METHOD PUBLIC Cycle // cyclic call for checking XtsStation state masks and command input from process
//-------------------------------------------------------------------------------------------------
//-------------------------------------------------------------------------------------------------
//  HAUD 2024 10 21
//  cyclic call required
//
//-------------------------------------------------------------------------------------------------
//-------------------------------------------------------------------------------------------------
// reference checks
//-------------------------------------------------------------------------------------------------
IF NOT __ISVALIDREF(_stControl)
THEN
  _eCheck                           := E_PROCESS_CHECK.REFERENCE_CTRL_INVALID;
  RETURN;
END_IF

IF NOT __ISVALIDREF(_stState)
THEN
  _eCheck                           := E_PROCESS_CHECK.REFERENCE_STATE_INVALID;
  RETURN;
END_IF
//-------------------------------------------------------------------------------------------------
//-------------------------------------------------------------------------------------------------
// plausibility checks
//-------------------------------------------------------------------------------------------------
IF NOT Check()
THEN
  // you shall not pass!!
  RETURN;
END_IF
//-------------------------------------------------------------------------------------------------
//-------------------------------------------------------------------------------------------------
// Message device identification
//-------------------------------------------------------------------------------------------------
_stMsg.eDevice                      := e_Device.Process + TO_UINT(_nProcessId);
//-------------------------------------------------------------------------------------------------
//-------------------------------------------------------------------------------------------------
// XtsStation states:
//  - fb_ProcessCollector extends fb_StationCollector: 
//    --> cyclic call of States() for getting station masks
//
//  - sets bit for every XtsStation
//-------------------------------------------------------------------------------------------------
//
States();                           // not just mental, literal
//-------------------------------------------------------------------------------------------------
//-------------------------------------------------------------------------------------------------
// process states
//-------------------------------------------------------------------------------------------------
CASE _stState.State
OF
  //-----------------------------------------------------------------------------------------------
  E_PROCESS_STATE.PROCESS_DISABLE:  // default wait state
    //-------------------------------------------------------------------------
    CASE _eStateProgress            // check if all my XtsStations are disabled
    OF
      E_PROGRESS.PROGRESS_INIT:
        IF (_wStateDisable = EXPT(2,_nStationCount)-1)                  // all stations in process range must be disabled at this point
        THEN
          // on a sunny afternoon, nothing to do, just sit and wait
          _eStateProgress           := E_PROGRESS.PROGRESS_BUSY;

          IF (_MessageLevel > E_MessageType.eMessageInfo)
          THEN
            _stMsg.eType            := E_MessageType.eMessageVerbose;
            _stMsg.eSubdevice       := e_Subdevice.Process_ProcessCollector_Cycle;
            _stMsg.iErrorNumber     := _wStateDisable;
            _stMsg.sText            := concat('_wStateDisable: ', BitsToString(_wStateDisable));
            _stMsg.sText            := concat(_stMsg.sText, ': ');
            _stMsg.sText            := concat(_stMsg.sText, TO_STRING(_eStateProgress));
            f_MessageSet(_stMsg);
          END_IF
        END_IF
    END_CASE
    //-------------------------------------------------------------------------
    CASE _eStateProgress            // check for process enable signal
    OF
      E_PROGRESS.PROGRESS_BUSY:
      CASE _stControl.Cmd                                               // check process command
      OF
        E_PROCESS_CTRL.PROCESS_ENABLE:                                  // only one thing to say here..
          _eCmd                     := _stControl.Cmd;                  // copy command from interface to local switch
          // you do what I say, when I say it
          _wActivateStation         := _stControl.ActivateStation;      // on enabling of process, copy my active stations from interface

          LogControl(_eCmd);

          _eStateProgress           := E_PROGRESS.PROGRESS_INIT;        // switch back sub state
          _stState.State            := E_PROCESS_STATE.PROCESS_ENABLE;  // switch to enable

          IF (_MessageLevel > E_MessageType.eMessageError)
          THEN
            _stMsg.eType            := E_MessageType.eMessageInfo;
            _stMsg.eSubdevice       := e_Subdevice.Process_ProcessCollector_Cycle;
            _stMsg.iErrorNumber     := _nProcessId;
            _stMsg.sText            := concat(TO_STRING(_stState.State), ': ');
            _stMsg.sText            := concat(_stMsg.sText, TO_STRING(_eStateProgress));
            f_MessageSet(_stMsg);
          END_IF
      END_CASE
    END_CASE
END_CASE
//-------------------------------------------------------------------------------------------------
//-------------------------------------------------------------------------------------------------
CASE _stState.State
OF
  //-----------------------------------------------------------------------------------------------
  E_PROCESS_STATE.PROCESS_ENABLE:   // wait here for process command "allow infeed"
    //-------------------------------------------------------------------------
    CASE _eStateProgress
    OF
      E_PROGRESS.PROGRESS_INIT:
        IF (_wStateEnable = _wActivateStation)                          // all active stations must be enabled
        THEN
          // we are truly equal, yet not the same
          _eStateProgress           := E_PROGRESS.PROGRESS_BUSY;

          IF (_MessageLevel > E_MessageType.eMessageInfo)
          THEN
            _stMsg.eType            := E_MessageType.eMessageVerbose;
            _stMsg.eSubdevice       := e_Subdevice.Process_ProcessCollector_Cycle;
            _stMsg.iErrorNumber     := _wStateEnable;
            _stMsg.sText            := concat('_wStateEnable: ', BitsToString(_wStateEnable));
            _stMsg.sText            := concat(_stMsg.sText, ': ');
            _stMsg.sText            := concat(_stMsg.sText, TO_STRING(_eStateProgress));
            f_MessageSet(_stMsg);
          END_IF
        END_IF
    END_CASE
    //-------------------------------------------------------------------------
    CASE _eStateProgress
    OF
      E_PROGRESS.PROGRESS_BUSY:
      // check command for further instructions
      CASE _stControl.Cmd
      OF
        E_PROCESS_CTRL.PROCESS_DISABLE:                                 // command decided to switch OFF  
          _eCmd                     := _stControl.Cmd;                  // copy command from interface

          LogControl(_eCmd);

          _eStateProgress           := E_PROGRESS.PROGRESS_INIT;        // switch back sub state
          _stState.State            := E_PROCESS_STATE.PROCESS_DISABLE;

          IF (_MessageLevel > E_MessageType.eMessageInfo)
          THEN
            _stMsg.eType            := E_MessageType.eMessageVerbose;
            _stMsg.eSubdevice       := e_Subdevice.Process_ProcessCollector_Cycle;
            _stMsg.iErrorNumber     := _nProcessId;
            _stMsg.sText            := concat(TO_STRING(_stState.State), ': ');
            _stMsg.sText            := concat(_stMsg.sText, TO_STRING(_eStateProgress));
            f_MessageSet(_stMsg);
          END_IF


        E_PROCESS_CTRL.PROCESS_STATIONS_INFEED,
        E_PROCESS_CTRL.PROCESS_STATIONS_ENTER,
        E_PROCESS_CTRL.PROCESS_STATIONS_SEND:                           // command decided to allow checking the infeed into process
          _eStateProgress           := E_PROGRESS.PROGRESS_INIT;        // switch back sub state
          _stState.State            := E_PROCESS_STATE.PROCESS_STATIONS_INFEED;

          IF (_MessageLevel > E_MessageType.eMessageWarning)
          THEN
            _stMsg.eType            := E_MessageType.eMessageInfo;
            _stMsg.eSubdevice       := e_Subdevice.Process_ProcessCollector_Cycle;
            _stMsg.iErrorNumber     := _nProcessId;
            _stMsg.sText            := concat(TO_STRING(_stState.State), ': ');
            _stMsg.sText            := concat(_stMsg.sText, TO_STRING(_eStateProgress));
            f_MessageSet(_stMsg);
          END_IF
      END_CASE
    END_CASE
END_CASE
//-------------------------------------------------------------------------------------------------
//-------------------------------------------------------------------------------------------------
CASE _stState.State
OF
  //-----------------------------------------------------------------------------------------------
  E_PROCESS_STATE.PROCESS_STATIONS_INFEED:  // wait state for checking infeed command
    //-------------------------------------------------------------------------
    CASE _eStateProgress
    OF
      E_PROGRESS.PROGRESS_INIT:
        IF (_wStateEnter = _wActivateStation)                           // all active XtsStations must have mover waiting
        THEN
          // mover IDs are known by now --> Check _nMoverIdQueue for your plausibility checks
          // master master, there's the thing I've been after
          _eStateProgress           := E_PROGRESS.PROGRESS_BUSY;

          IF (_MessageLevel > E_MessageType.eMessageInfo)
          THEN
            _stMsg.eType            := E_MessageType.eMessageVerbose;
            _stMsg.eSubdevice       := e_Subdevice.Process_ProcessCollector_Cycle;
            _stMsg.iErrorNumber     := _wStateEnter;
            _stMsg.sText            := concat('_wStateEnter: ', BitsToString(_wStateEnter));
            _stMsg.sText            := concat(_stMsg.sText, ': ');
            _stMsg.sText            := concat(_stMsg.sText, TO_STRING(_eStateProgress));
            f_MessageSet(_stMsg);
          END_IF
        END_IF
    END_CASE
    //-------------------------------------------------------------------------
    CASE _eStateProgress
    OF
      E_PROGRESS.PROGRESS_BUSY:
      CASE _stControl.Cmd                                               // check command from interface
      OF
        E_PROCESS_CTRL.PROCESS_STATIONS_ENTER:
          _eCmd                     := _stControl.Cmd;                  // copy command to start infeed of movers

          LogControl(_eCmd);

          _eStateProgress           := E_PROGRESS.PROGRESS_INIT;        // switch back sub state
          _stState.State            := E_PROCESS_STATE.PROCESS_START;

          IF (_MessageLevel > E_MessageType.eMessageError)
          THEN
            _stMsg.eType            := E_MessageType.eMessageInfo;
            _stMsg.eSubdevice       := e_Subdevice.Process_ProcessCollector_Cycle;
            _stMsg.iErrorNumber     := _nProcessId;
            _stMsg.sText            := concat(TO_STRING(_stState.State), ': ');
            _stMsg.sText            := concat(_stMsg.sText, TO_STRING(_eStateProgress));
            f_MessageSet(_stMsg);
          END_IF


        E_PROCESS_CTRL.PROCESS_STATIONS_SEND:
          _eCmd                     := _stControl.Cmd;                  // start skipping of process

          LogControl(_eCmd);

          _eStateProgress           := E_PROGRESS.PROGRESS_INIT;        // switch back sub state
          _stState.State            := E_PROCESS_STATE.PROCESS_STATIONS_OUTFEED;

          IF (_MessageLevel > E_MessageType.eMessageError)
          THEN
            _stMsg.eType            := E_MessageType.eMessageInfo;
            _stMsg.eSubdevice       := e_Subdevice.Process_ProcessCollector_Cycle;
            _stMsg.iErrorNumber     := _nProcessId;
            _stMsg.sText            := concat(TO_STRING(_stState.State), ': ');
            _stMsg.sText            := concat(_stMsg.sText, TO_STRING(_eStateProgress));
            f_MessageSet(_stMsg);
          END_IF
      END_CASE
    END_CASE
END_CASE
//-------------------------------------------------------------------------------------------------
//-------------------------------------------------------------------------------------------------
CASE _stState.State
OF
  //-----------------------------------------------------------------------------------------------
  E_PROCESS_STATE.PROCESS_STATIONS_NEST:  // wait state before movers are positioned to next nest
    //-------------------------------------------------------------------------
    CASE _eStateProgress
    OF
      E_PROGRESS.PROGRESS_INIT:
        IF (_wStateNest = _wActivateStation)  // ...to include everyone
        THEN
          _eStateProgress           := E_PROGRESS.PROGRESS_BUSY;

          IF (_MessageLevel > E_MessageType.eMessageWarning)
          THEN
            _stMsg.eType            := E_MessageType.eMessageInfo;
            _stMsg.eSubdevice       := e_Subdevice.Process_ProcessCollector_Cycle;
            _stMsg.iErrorNumber     := _wStateNest;
            _stMsg.sText            := concat('_wStateNest: ', BitsToString(_wStateNest));
            _stMsg.sText            := concat(_stMsg.sText, ': ');
            _stMsg.sText            := concat(_stMsg.sText, TO_STRING(_eStateProgress));
            f_MessageSet(_stMsg);
          END_IF
        END_IF
    END_CASE
    //-------------------------------------------------------------------------
    CASE _eStateProgress
    OF
      E_PROGRESS.PROGRESS_BUSY:
      CASE _stControl.Cmd
      OF
        E_PROCESS_CTRL.PROCESS_STATIONS_ENTER:
          _eCmd                     := _stControl.Cmd;                  // copy command to start movement to next nest

          LogControl(_eCmd);

          _eStateProgress           := E_PROGRESS.PROGRESS_INIT;        // switch back sub state
          _stState.State            := E_PROCESS_STATE.PROCESS_START;

          IF (_MessageLevel > E_MessageType.eMessageWarning)
          THEN
            _stMsg.eType            := E_MessageType.eMessageInfo;
            _stMsg.eSubdevice       := e_Subdevice.Process_ProcessCollector_Cycle;
            _stMsg.iErrorNumber     := _nProcessId;
            _stMsg.sText            := concat(TO_STRING(_stState.State), ': ');
            _stMsg.sText            := concat(_stMsg.sText, TO_STRING(_eStateProgress));
            f_MessageSet(_stMsg);
          END_IF
      END_CASE
    END_CASE
END_CASE
//-------------------------------------------------------------------------------------------------
//-------------------------------------------------------------------------------------------------
CASE _stState.State
OF
  //-----------------------------------------------------------------------------------------------
  E_PROCESS_STATE.PROCESS_START:    // wait state for movers to arrive
    //-------------------------------------------------------------------------
    CASE _eStateProgress
    OF
      E_PROGRESS.PROGRESS_INIT:
        IF (_wStateStart = _wActivateStation)  
          // all active XtsStations have mover in standstill after infeed, 
          // process handshake may now start
        THEN
          // movers have arrived and are in standstill
          _eStateProgress           := E_PROGRESS.PROGRESS_BUSY;

          IF (_MessageLevel > E_MessageType.eMessageInfo)
          THEN
            _stMsg.eType            := E_MessageType.eMessageVerbose;
            _stMsg.eSubdevice       := e_Subdevice.Process_ProcessCollector_Cycle;
            _stMsg.iErrorNumber     := _wStateStart;
            _stMsg.sText            := concat('_wStateStart: ', BitsToString(_wStateStart));
            _stMsg.sText            := concat(_stMsg.sText, ': ');
            _stMsg.sText            := concat(_stMsg.sText, TO_STRING(_eStateProgress));
            f_MessageSet(_stMsg);
          END_IF
        END_IF
    END_CASE
    //-------------------------------------------------------------------------
    CASE _eStateProgress
    OF
      E_PROGRESS.PROGRESS_BUSY:
      CASE _stControl.Cmd
      OF
        E_PROCESS_CTRL.PROCESS_START,
        E_PROCESS_CTRL.PROCESS_DONE,
        E_PROCESS_CTRL.PROCESS_STATIONS_OUTFEED:
          _eCmd                     := E_PROCESS_CTRL.PROCESS_DONE;     // first handshake for starting process

          LogControl(_eCmd);

          _eStateProgress           := E_PROGRESS.PROGRESS_INIT;        // switch back sub state
          _stState.State            := E_PROCESS_STATE.PROCESS_DONE;

          IF (_MessageLevel > E_MessageType.eMessageWarning)
          THEN
            _stMsg.eType            := E_MessageType.eMessageInfo;
            _stMsg.eSubdevice       := e_Subdevice.Process_ProcessCollector_Cycle;
            _stMsg.iErrorNumber     := _nProcessId;
            _stMsg.sText            := concat(TO_STRING(_stState.State), ': ');
            _stMsg.sText            := concat(_stMsg.sText, TO_STRING(_eStateProgress));
            f_MessageSet(_stMsg);
          END_IF
      END_CASE
    END_CASE
END_CASE
//-------------------------------------------------------------------------------------------------
//-------------------------------------------------------------------------------------------------
CASE _stState.State
OF
  E_PROCESS_STATE.PROCESS_DONE:     // wait state for process done
    //-------------------------------------------------------------------------
    CASE _eStateProgress
    OF
      E_PROGRESS.PROGRESS_INIT:
        IF (_wStateDone = _wActivateStation)
        THEN
          // first handshake done
          _eStateProgress           := E_PROGRESS.PROGRESS_BUSY;

          IF (_MessageLevel > E_MessageType.eMessageInfo)
          THEN
            _stMsg.eType            := E_MessageType.eMessageVerbose;
            _stMsg.eSubdevice       := e_Subdevice.Process_ProcessCollector_Cycle;
            _stMsg.iErrorNumber     := _wStateDone;
            _stMsg.sText            := concat('_wStateDone: ', BitsToString(_wStateDone));
            _stMsg.sText            := concat(_stMsg.sText, ': ');
            _stMsg.sText            := concat(_stMsg.sText, TO_STRING(_eStateProgress));
            f_MessageSet(_stMsg);
          END_IF
        END_IF
    END_CASE
    //-------------------------------------------------------------------------
    CASE _eStateProgress
    OF
      E_PROGRESS.PROGRESS_BUSY:
      CASE _stControl.Cmd
      OF
        E_PROCESS_CTRL.PROCESS_DONE,
        E_PROCESS_CTRL.PROCESS_STATIONS_OUTFEED:
          _eCmd                     := _stControl.Cmd;                  // second handshake for finishing process

          LogControl(_eCmd);

          _eStateProgress           := E_PROGRESS.PROGRESS_CHECK;       // check mover after process done
      END_CASE
    //-------------------------------------------------------------------------
      E_PROGRESS.PROGRESS_CHECK:
        IF (_wStateNest > 0)        // mover has to be worked again
        THEN
          _eStateProgress           := E_PROGRESS.PROGRESS_INIT;        // switch back sub state
          _stState.State            := E_PROCESS_STATE.PROCESS_STATIONS_NEST;

          IF (_MessageLevel > E_MessageType.eMessageInfo)
          THEN
            _stMsg.eType            := E_MessageType.eMessageVerbose;
            _stMsg.eSubdevice       := e_Subdevice.Process_ProcessCollector_Cycle;
            _stMsg.iErrorNumber     := _nProcessId;
            _stMsg.sText            := concat(TO_STRING(_stState.State), ': ');
            _stMsg.sText            := concat(_stMsg.sText, TO_STRING(_eStateProgress));
            f_MessageSet(_stMsg);
          END_IF

        ELSIF (_wStateOut > 0)      // mover has to leave
        THEN
          _eStateProgress           := E_PROGRESS.PROGRESS_INIT;        // switch back sub state
          _stState.State            := E_PROCESS_STATE.PROCESS_STATIONS_OUTFEED;

          IF (_MessageLevel > E_MessageType.eMessageInfo)
          THEN
            _stMsg.eType            := E_MessageType.eMessageVerbose;
            _stMsg.eSubdevice       := e_Subdevice.Process_ProcessCollector_Cycle;
            _stMsg.iErrorNumber     := _nProcessId;
            _stMsg.sText            := concat(TO_STRING(_stState.State), ': ');
            _stMsg.sText            := concat(_stMsg.sText, TO_STRING(_eStateProgress));
            f_MessageSet(_stMsg);
          END_IF
        END_IF
    END_CASE
END_CASE
//-------------------------------------------------------------------------------------------------
//-------------------------------------------------------------------------------------------------
CASE _stState.State
OF
  E_PROCESS_STATE.PROCESS_STATIONS_OUTFEED:   // wait state before movers are sent out
    //-------------------------------------------------------------------------
    CASE _eStateProgress
    OF
      E_PROGRESS.PROGRESS_INIT:
        IF (_wStateOut = _wActivateStation)
        THEN
          // all active stations want to send out mover
          // now is the time for you to have decided the TargetStation(s) and TargetMask(s)
          _eStateProgress           := E_PROGRESS.PROGRESS_BUSY;

          IF (_MessageLevel > E_MessageType.eMessageInfo)
          THEN
            _stMsg.eType            := E_MessageType.eMessageVerbose;
            _stMsg.eSubdevice       := e_Subdevice.Process_ProcessCollector_Cycle;
            _stMsg.iErrorNumber     := _wStateOut;
            _stMsg.sText            := concat('_wStateOut: ', BitsToString(_wStateOut));
            _stMsg.sText            := concat(_stMsg.sText, ': ');
            _stMsg.sText            := concat(_stMsg.sText, TO_STRING(_eStateProgress));
            f_MessageSet(_stMsg);
          END_IF
        END_IF
    END_CASE
    //-------------------------------------------------------------------------
    CASE _eStateProgress
    OF
      E_PROGRESS.PROGRESS_BUSY:     // now is the time to get/write target data
      CASE _stControl.Cmd
      OF
        E_PROCESS_CTRL.PROCESS_STATIONS_OUTFEED:  // before you start the outfeed of station, get/write target data on the outside. Use properties: TargetIndex; TargetMask
          _eCmd                     := _stControl.Cmd;

          LogControl(_eCmd);

          _eStateProgress           := E_PROGRESS.PROGRESS_CHECK;       // check movers gone

          IF (_MessageLevel > E_MessageType.eMessageError)
          THEN
            _stMsg.eType            := E_MessageType.eMessageInfo;
            _stMsg.eSubdevice       := e_Subdevice.Process_ProcessCollector_Cycle;
            _stMsg.iErrorNumber     := _nProcessId;
            _stMsg.sText            := concat(TO_STRING(_stState.State), ': ');
            _stMsg.sText            := concat(_stMsg.sText, TO_STRING(_eStateProgress));
            f_MessageSet(_stMsg);
          END_IF
      END_CASE
    END_CASE
    //-------------------------------------------------------------------------
    CASE _eStateProgress
    OF
      E_PROGRESS.PROGRESS_CHECK:
        IF (_wStateOut = 0)         // all stations are empty, go back to start new infeed of movers
        THEN
          _eStateProgress           := E_PROGRESS.PROGRESS_INIT;        // switch back sub state
          _stState.State            := E_PROCESS_STATE.PROCESS_DISABLE; // switch back to disabled state

          IF (_MessageLevel > E_MessageType.eMessageInfo)
          THEN
            _stMsg.eType            := E_MessageType.eMessageVerbose;
            _stMsg.eSubdevice       := e_Subdevice.Process_ProcessCollector_Cycle;
            _stMsg.iErrorNumber     := _wStateOut;
            _stMsg.sText            := concat('_wStateOut: ', BitsToString(_wStateOut));
            _stMsg.sText            := concat(_stMsg.sText, ': ');
            _stMsg.sText            := concat(_stMsg.sText, TO_STRING(_eStateProgress));
            f_MessageSet(_stMsg);
          END_IF
        END_IF
    END_CASE
END_CASE
//-------------------------------------------------------------------------------------------------
// _eStateProgress information to process result
//-------------------------------------------------------------------------------------------------
_stState.Result                     := _eStateProgress;
//-------------------------------------------------------------------------------------------------
//-------------------------------------------------------------------------------------------------
// _eCheck information for plausibility checks
//-------------------------------------------------------------------------------------------------
_stState.Check                      := _eCheck;
//-------------------------------------------------------------------------------------------------
//-------------------------------------------------------------------------------------------------
// _eCmd - command switch
//-------------------------------------------------------------------------------------------------
Controls(_eCmd);                    // cyclic call for setting commands on XtsStations in process range
//-------------------------------------------------------------------------------------------------
//-------------------------------------------------------------------------------------------------
END_METHOD

METHOD PUBLIC Init : E_PROGRESS // clears all XtsSubstations, then disables all
VAR_INPUT
  Execute     : BOOL;
END_VAR
VAR_INST
  _nIndexStation        : UINT;
  _nErrorId             : UDINT;
  _eState               : E_PROGRESS;
END_VAR
//-----------------------------------------------------------------------------
IF NOT Execute 
THEN 
	_eState                       := E_PROGRESS.PROGRESS_INIT; 
END_IF 
//-----------------------------------------------------------------------------
IF NOT Check() 
THEN 
	Init                          := E_PROGRESS.PROGRESS_ERROR; 
	RETURN; 
END_IF
//-----------------------------------------------------------------------------
//-----------------------------------------------------------------------------
CASE _eState
OF
  E_PROGRESS.PROGRESS_INIT:
    IF Execute
    THEN
      _nIndexStation            := _nStationLast;
      _nErrorId                 := 0;
      _eState                   := E_PROGRESS.PROGRESS_BUSY;
      memset(ADR(_wTargetMask), 1, SIZEOF(_wTargetMask));

      _eCmd                     := E_PROCESS_CTRL.PROCESS_INIT;
      _stState.State            := E_PROCESS_STATE.PROCESS_INVALID;
      _eStateProgress           := E_PROGRESS.PROGRESS_INVALID;


      _stMsg.eType              := _MessageLevel;

      IF (_MessageLevel = E_MessageType.eMessageVerbose)
      THEN
        _stMsg.eSubdevice       := e_Subdevice.Process_ProcessCollector_Init;
        _stMsg.iErrorNumber     := _nIndexStation;
        _stMsg.sText            := concat('.Init: ', TO_STRING(_eState));
        f_MessageSet(_stMsg);
      END_IF
    END_IF
END_CASE
//-----------------------------------------------------------------------------
//-----------------------------------------------------------------------------
CASE _eState
OF
  E_PROGRESS.PROGRESS_BUSY:
    _stStationCtrl[_nIndexStation].Cmd     := E_STATION_CTRL.STATION_INIT;
    _eState                     := E_PROGRESS.PROGRESS_PREPARE;

    IF (_MessageLevel = E_MessageType.eMessageVerbose)
    THEN
      _stMsg.eSubdevice         := e_Subdevice.Process_ProcessCollector_Init;
      _stMsg.iErrorNumber       := _nIndexStation;
      _stMsg.sText              := concat(TO_STRING(_stStationCtrl[_nIndexStation].Cmd), ': ');
      _stMsg.sText              := concat(_stMsg.sText, TO_STRING(_eState));
      f_MessageSet(_stMsg);
    END_IF

  E_PROGRESS.PROGRESS_PREPARE:
    IF (_nIndexStation < _nStationFirst+1)
    THEN
      _eCmdOld                  :=
      _eCmd                     := E_PROCESS_CTRL.PROCESS_DISABLE;
      _nIndexStation            := _nStationFirst;
      _eState                   := E_PROGRESS.PROGRESS_STARTUP;
    ELSE
      IF (_stStationState[_nIndexStation].State = E_STATION_STATE.STATION_INIT)
      THEN
        _nIndexStation          := _nIndexStation - 1;
        _eState                 := E_PROGRESS.PROGRESS_BUSY;
      ELSE
        _eState                 := E_PROGRESS.PROGRESS_BUSY;
      END_IF
    END_IF

  E_PROGRESS.PROGRESS_STARTUP:
    _stStationCtrl[_nIndexStation].Cmd     := E_STATION_CTRL.STATION_DISABLE;
    _eState                     := E_PROGRESS.PROGRESS_CHECK;

    IF (_MessageLevel = E_MessageType.eMessageVerbose)
    THEN
      _stMsg.eSubdevice         := e_Subdevice.Process_ProcessCollector_Init;
      _stMsg.iErrorNumber       := _nIndexStation;
      _stMsg.sText              := concat(TO_STRING(_stStationCtrl[_nIndexStation].Cmd), ': ');
      _stMsg.sText              := concat(_stMsg.sText, TO_STRING(_eState));
      f_MessageSet(_stMsg);
    END_IF

  E_PROGRESS.PROGRESS_CHECK:
    IF NOT (_nIndexStation > _nStationLast-1)
    THEN
      IF (_stStationState[_nIndexStation].State = E_STATION_STATE.STATION_DISABLE)
      THEN
        _nIndexStation          := _nIndexStation + 1;
        _eState                 := E_PROGRESS.PROGRESS_STARTUP;
      END_IF
    ELSE
      // give back result
      _eState                   := E_PROGRESS.PROGRESS_DONE;

      // where were I?
      IF (_MessageLevel = E_MessageType.eMessageVerbose)
      THEN
        _stMsg.eSubdevice       := e_Subdevice.Process_ProcessCollector_Init;
        _stMsg.iErrorNumber     := _nProcessId;
        _stMsg.sText            := concat('.Clear: ', TO_STRING(_stState.State));
        f_MessageSet(_stMsg);
      END_IF

      // clear Cycle() state machine
      _stState.State            := E_PROCESS_STATE.PROCESS_DISABLE;
      _eStateProgress           := E_PROGRESS.PROGRESS_INIT;

      IF (_MessageLevel = E_MessageType.eMessageVerbose)
      THEN
        // init done
        _stMsg.eSubdevice       := e_Subdevice.Process_ProcessCollector_Init;
        _stMsg.iErrorNumber     := _nProcessId;
        _stMsg.sText            := concat('.Init: ', TO_STRING(_eState));
        f_MessageSet(_stMsg);
      END_IF
    END_IF
END_CASE
//-----------------------------------------------------------------------------
//-----------------------------------------------------------------------------

Init := _eState;
END_METHOD

METHOD PRIVATE LogControl
VAR_INPUT
  Cmd         : E_PROCESS_CTRL;
END_VAR
IF (Cmd <> _eCmdOld)
THEN
  IF (_MessageLevel > E_MessageType.eMessageWarning)
  THEN
    _stMsg.eType                          := E_MessageType.eMessageInfo;
    _stMsg.eSubdevice                     := e_Subdevice.Process_ProcessCollector_Control;
    _stMsg.iErrorNumber                   := _nProcessId;
    _stMsg.sText                          := 'Cmd: ';
    _stMsg.sText                          := concat(_stMsg.sText, TO_STRING(Cmd));
    f_MessageSet(_stMsg);
  END_IF

  CASE Cmd                                               // check process command
  OF
    E_PROCESS_CTRL.PROCESS_ENABLE:
      IF (_MessageLevel = E_MessageType.eMessageVerbose)
      THEN
        _stMsg.eType                      := E_MessageType.eMessageVerbose;
        _stMsg.eSubdevice                 := e_Subdevice.Process_ProcessCollector_Control;
        _stMsg.iErrorNumber               := _wActivateStation;
        _stMsg.sText                      := concat('_wActivateStation: ', BitsToString(_wActivateStation));
        f_MessageSet(_stMsg);
      END_IF
   END_CASE
  _eCmdOld                                := Cmd;
END_IF
END_METHOD

PROPERTY MessageLevel : e_MessageType
GET
MessageLevel := _MessageLevel;
END_GET
SET
VAR
  _ix : uint;
END_VAR
_MessageLevel := MessageLevel;

IF NOT (_eCheck = E_PROCESS_CHECK.CHECK_DONE)
THEN
  RETURN;
ELSE
  FOR _ix := _nStationFirst TO _nStationLast
  DO
    GVL_MSG_XTS.MessageLevelStations[_ix]   := _MessageLevel;
  END_FOR
END_IF
END_SET
END_PROPERTY

PROPERTY MoverCountTotal : udint
GET
MoverCountTotal := _nMoverCountTotal;
END_GET
END_PROPERTY

PROPERTY MoverPerMinute : udint
GET
MoverPerMinute := _AllStationMoverPerMinute;
END_GET
END_PROPERTY

PROPERTY ProcessCtrl : reference to st_process_ctrl
GET
ProcessCtrl REF= _stControl;
END_GET
SET
_stControl ref= ProcessCtrl;
END_SET
END_PROPERTY

PROPERTY ProcessId : E_INSTANCE
GET
Processid := _nProcessId;
END_GET
SET
_nProcessId := ProcessId;
END_SET
END_PROPERTY

PROPERTY ProcessState : reference to st_process_state
GET
ProcessState REF= _stState;
END_GET
SET
_stState ref= ProcessState;
END_SET
END_PROPERTY

PROPERTY TargetIndex : ARRAY[1..SIZEOF(T_PROCESS)*8] OF USINT
GET
TargetIndex := _nTargetIndex;
END_GET
SET
_nTargetIndex := TargetIndex;
END_SET
END_PROPERTY

PROPERTY TargetMask : ARRAY[1..SIZEOF(T_PROCESS)*8] OF BYTE
GET
TargetMask := _wTargetMask;
END_GET
SET
_wTargetMask := TargetMask;
END_SET
END_PROPERTY

METHOD Template : E_PROGRESS
VAR_INPUT
  Execute     : BOOL;
END_VAR
VAR_INST
  _nErrorId   : UDINT;
  _eState     : E_PROGRESS;
END_VAR
//-----------------------------------------------------------------------------
IF NOT Execute 
THEN 
	_eState                       := E_PROGRESS.PROGRESS_INIT; 
END_IF 
//-----------------------------------------------------------------------------
IF NOT Check() 
THEN 
	Template_1                    := E_PROGRESS.PROGRESS_ERROR; 
	RETURN; 
END_IF
//-----------------------------------------------------------------------------
//-----------------------------------------------------------------------------
CASE _eState
OF
  E_PROGRESS.PROGRESS_INIT:
    IF Execute
    THEN
      _nErrorId                 := 0;

      _eState                   := E_PROGRESS.PROGRESS_BUSY;
    END_IF
END_CASE
//-----------------------------------------------------------------------------
//-----------------------------------------------------------------------------
CASE _eState
OF
  E_PROGRESS.PROGRESS_BUSY:
    _eState                     := E_PROGRESS.PROGRESS_PREPARE;
END_CASE
//-----------------------------------------------------------------------------
//-----------------------------------------------------------------------------
CASE _eState
OF
  E_PROGRESS.PROGRESS_PREPARE:

    IF (.Error)
    THEN
      _eState                   := E_PROGRESS.PROGRESS_ERROR;
      _nErrorId                 := 


    ELSIF (.Done)
    THEN
      _eState                   := E_PROGRESS.;

    END_IF
END_CASE
//-----------------------------------------------------------------------------
//-----------------------------------------------------------------------------

Template_1                      := _eState;
END_METHOD

END_FUNCTION_BLOCK

// ---- APPLICATION/_types/Collector/fb_StationCollector.TcPOU
//---------------------------------------------------------------------------------------------------------------
//
//  HAUD 2024.10.13
//
//
//  fb_StateCollector
//  - base class for process handling
//  - collects states from range of XtsStations
//
//---------------------------------------------------------------------------------------------------------------//
// This SOFTWARE is provided as an Example by THE PROVIDER "as is" and "with all faults." THE PROVIDER makes no  //
// representations or warranties of any kind concerning the safety, suitability, lack of viruses, inaccuracies,  //
// typographical errors, or other harmful components of this SOFTWARE. There are inherent dangers in the use of  //
// any software, and you are solely responsible for determining whether this SOFTWARE is compatible with your    //
// equipment and other software installed on your equipment. You are also solely responsible for the protection  //
// of your equipment and backup of your data, and THE PROVIDER will not be liable for any damages you may suffer //
// in connection with using, modifying, or distributing this SOFTWARE.                                           //
//---------------------------------------------------------------------------------------------------------------//
FUNCTION_BLOCK ABSTRACT fb_StationCollector
VAR
  {info ' extend/add enum members to E_INSTANCE as you need them '}
  _nProcessId     : E_INSTANCE; // whoami

  _eCheck             : E_PROCESS_CHECK;
  _nStationCount      : UINT;

  _nStationFirst,
  _nStationLast       : UINT; // closed range of XtsStations

  // ctrl / state datafields for extern control
  _stStationCtrl      : REFERENCE TO ARRAY[1..MAX_STATION] OF ST_STATION_CTRL;   // control for extern to write
  _stStationState     : REFERENCE TO ARRAY[1..MAX_STATION] OF ST_STATION_STATE;  // state for extern to read

  // mover info datafield
  _MoverInfo          : REFERENCE TO ARRAY[1..MAX_MOVER] OF ST_MOVER_INFO;

  // One Process    - multiple XtsStations
  // One XtsStation - One Mover
  //
  // state words for XtsStations in my range
  {attribute 'displaymode':='bin'}
  _wStateDisable      : T_PROCESS;
  {attribute 'displaymode':='bin'}
  _wStateEnable       : T_PROCESS;
  {attribute 'displaymode':='bin'}
  _wStateEnter        : T_PROCESS;
  {attribute 'displaymode':='bin'}
  _wStateStart        : T_PROCESS;
  {attribute 'displaymode':='bin'}
  _wStateDone         : T_PROCESS;
  {attribute 'displaymode':='bin'}
  _wStateNest         : T_PROCESS;
  {attribute 'displaymode':='bin'}
  _wStateOut          : T_PROCESS;
  {attribute 'displaymode':='bin'}
  _wStateGone         : T_PROCESS;
  {attribute 'displaymode':='bin'}
  _wError             : T_PROCESS;
  {attribute 'displaymode':='bin'}
  _wErrorFatal        : T_PROCESS;

  // One Process    - multiple XtsStations
  // One XtsStation - One Mover
  //

  // important state infos from XtsStations
  _nMoverIdQueue,
  _nStationQueue              : ARRAY[1..SIZEOF(T_PROCESS)*8] OF UINT; // single queues from sub stations
  _nProcessQueue              : UINT; // sum of all sub station queues

  _AllStationMoverPerMinute   : UINT;
  _tonPartsPerMinute          : Tc2_Standard.TON;

  _nMoverCountTotal           : UDINT;

  _stMsg                      : ST_Message;
  _MessageLevel               : E_MessageType;
END_VAR

METHOD PUBLIC BitDel : T_PROCESS
VAR_INPUT
  inVal   : T_PROCESS;
  bitNo   : DINT;
END_VAR
VAR
  wConst : T_PROCESS := 1;
END_VAR
IF ( inVal AND SHL( wConst,TO_SINT(bitNo) MOD TO_INT(SIZEOF(T_PROCESS)*8) ) ) > 0 THEN
  BitDel := inVal XOR (SHL( wConst,TO_SINT(bitNo) MOD TO_INT(SIZEOF(T_PROCESS)*8) ));
ELSE
  BitDel := inVal;
END_IF
END_METHOD

METHOD PUBLIC BitGet : BOOL
VAR_INPUT
  inVal   : T_PROCESS;
  bitNo   : DINT;
END_VAR
VAR
  wConst : T_PROCESS := 1;
END_VAR
IF ( inVal AND SHL( wConst,TO_SINT(bitNo) MOD TO_INT(SIZEOF(T_PROCESS)*8) ) ) > 0
THEN
  BitGet := TRUE;
ELSE
  BitGet := FALSE;
END_IF
END_METHOD

METHOD PUBLIC BitSet : T_PROCESS
VAR_INPUT
  inVal   : T_PROCESS;
  bitNo   : DINT;
END_VAR
VAR
  wConst  : T_PROCESS := 1;
END_VAR
BitSet := inVal OR SHL( wConst,TO_SINT(bitNo) MOD TO_INT(SIZEOF(T_PROCESS)*8) );
END_METHOD

METHOD BitsToString : STRING(SIZEOF(T_PROCESS)*8) // T_PROCESS to string
VAR_INPUT
  inVal       : T_PROCESS;
END_VAR
VAR
  _nx         : DINT;
  _str        : STRING(SIZEOF(T_PROCESS)*8);
END_VAR
FOR _nx := ((SIZEOF(inVal)*8)) TO 1 BY(-1)
DO
  IF (BitGet(inVal, _nx-1))
  THEN
    _str     := concat(_str, '1');
  ELSE
    _str     := concat(_str, '0');
  END_IF
END_FOR

BitsToString := _str;
END_METHOD

METHOD Check : BOOL
VAR_INPUT
END_VAR

IF NOT (_nStationLast > 0)
THEN
  _eCheck             := E_PROCESS_CHECK.STATION_LAST_ZERO;
  RETURN;
END_IF

IF NOT (_nStationFirst > 0)
THEN
  _eCheck             := E_PROCESS_CHECK.STATION_FIRST_ZERO;

  _stMsg.eType        := E_MessageType.eMessageWarning;
  _stMsg.eSubdevice   := e_Subdevice.Process_StationCollector;
  _stMsg.sText        := TO_STRING(_eCheck);
  f_MessageSet(_stMsg);

  _nStationFirst      := _nStationLast;
END_IF

IF NOT (_nStationLast < MAX_STATION+1)
THEN
  _eCheck         := E_PROCESS_CHECK.STATION_LAST_MAX;
  RETURN;
END_IF

IF NOT (_nStationFirst < MAX_STATION+1)
THEN
  _eCheck         := E_PROCESS_CHECK.STATION_FIRST_MAX;
  RETURN;
END_IF

_nStationCount    := _nStationLast - _nStationFirst + 1;
IF NOT (_nStationCount > 0)
THEN
  _eCheck         := E_PROCESS_CHECK.STATION_COUNT_NEGATIVE;
  RETURN;
END_IF

IF (_nStationCount > SIZEOF(T_PROCESS)*8)
THEN
  _eCheck         := E_PROCESS_CHECK.STATION_COUNT_TOO_HIGH;
  RETURN;
END_IF
//-------------------------------------------------------------------------------------------------
// reference checks
//-------------------------------------------------------------------------------------------------
IF NOT __ISVALIDREF(_MoverInfo)
THEN
  _eCheck         := E_PROCESS_CHECK.REFERENCE_MOVER_INFO_INVALID;
  RETURN;
END_IF

_eCheck           := E_PROCESS_CHECK.CHECK_DONE;
Check             := TRUE;
END_METHOD

METHOD GetMoverInStation : ST_MOVER_INFO // mover in station info
VAR_INPUT
  nStation            : UINT;   // index of GVL_XTS.StationState[nStation]
END_VAR
IF NOT Check() THEN RETURN; END_IF

IF NOT (nStation > 0) OR
   NOT (nStation < MAX_STATION+1)
THEN
  RETURN;
ELSE
  IF NOT (_stStationState[nStation].nMoverId > 0)
  THEN
    RETURN;
  ELSE
    GetMoverInStation           := _MoverInfo[_stStationState[nStation].nMoverId];
  END_IF
END_IF
END_METHOD

METHOD GetStationState : ST_STATION_STATE
VAR_INPUT
  nStation            : UINT;   // index of GVL_XTS.StationState[nStation]
END_VAR
IF NOT Check() THEN RETURN; END_IF

IF NOT (nStation > 0) OR
   NOT (nStation < MAX_STATION+1)
THEN
  RETURN;
ELSE
  GetStationState               := _stStationState[nStation];
END_IF
END_METHOD

PROPERTY MoverInfo : REFERENCE TO ARRAY[1..MAX_MOVER] OF ST_MOVER_INFO
SET
_MoverInfo REF= MoverInfo;
END_SET
END_PROPERTY

PROPERTY QueueMoverIDs : ARRAY[1..SIZEOF(T_PROCESS)*8] OF UINT
GET
QueueMoverIDs := _nMoverIdQueue;
END_GET
END_PROPERTY

PROPERTY QueueProcessCount : UINT // sum of all station queues
GET
QueueProcessCount := _nProcessQueue;
END_GET
END_PROPERTY

PROPERTY QueueStationCount : ARRAY[1..SIZEOF(T_PROCESS)*8] OF UINT
GET
QueueStationCount := _nStationQueue;
END_GET
END_PROPERTY

METHOD PROTECTED States // cyclic call for collecting XtsStation state masks
VAR_INST
  _idx    	: UINT;
  _k                    : UINT;
  _rtrigProcess         : ARRAY[1..MAX_STATION] OF Tc2_Standard.R_TRIG;
  _rtrigProcessEnter    : ARRAY[1..MAX_STATION] OF Tc2_Standard.R_TRIG;
  _rtrigProcessStart    : ARRAY[1..MAX_STATION] OF Tc2_Standard.R_TRIG;

  _nMoverPerMinute,
  _nMoverCount,
  _nMoverCountOld       : ARRAY[1..MAX_STATION]  OF UINT;

  _nMoverCountEnter,
  _nMoverCountEnterOld  : ARRAY[1..MAX_STATION]  OF UINT;

  _nMoverCountStart,
  _nMoverCountStartOld  : ARRAY[1..MAX_STATION]  OF UINT;


  _interAllStationsCounter    : UINT;
END_VAR
//-------------------------------------------------------------------------------------------------
//-------------------------------------------------------------------------------------------------
//  HAUD 2024 10 21
//  cyclic call must be implemented by inheriting class 
//  one bit in masks for every XtsStation in process
//
//-------------------------------------------------------------------------------------------------
//-------------------------------------------------------------------------------------------------
_wError                     :=
_wErrorFatal                := 0;

// the sum of movers waiting
_nProcessQueue              := 0;   // calc every plc cycle (see below)

// range checks of _nStationFirst; _nStationLast
IF NOT Check()
THEN
  RETURN;
END_IF

FOR _idx := _nStationLast TO _nStationFirst BY(-1)
DO
  // copy queue for every XtsStation to local for readability (debugging)
  _nStationQueue[(_idx-_nStationFirst+1)] := _stStationState[_idx].nQueue;

  // calc sum of queues for process
  _nProcessQueue                          := _nProcessQueue + _stStationState[_idx].nQueue;

  // get mover ID for all XtsStations in range
  _nMoverIdQueue[(_idx-_nStationFirst+1)] := _stStationState[_idx].nMoverId;

  CASE _stStationCtrl[_idx].Cmd
  OF
    E_STATION_CTRL.STATION_INIT:
      _wStateDisable        := BitDel(_wStateDisable,(_idx - _nStationFirst));
      _wStateEnable         := BitDel(_wStateEnable, (_idx - _nStationFirst));
      _wStateEnter          := BitDel(_wStateEnter,  (_idx - _nStationFirst));
      _wStateStart          := BitDel(_wStateStart,  (_idx - _nStationFirst));
      _wStateDone           := BitDel(_wStateDone,   (_idx - _nStationFirst));
      _wStateNest           := BitDel(_wStateNest,   (_idx - _nStationFirst));
      _wStateOut            := BitDel(_wStateOut,    (_idx - _nStationFirst));
      _wStateGone           := BitDel(_wStateGone,   (_idx - _nStationFirst));
  END_CASE

  CASE _stStationState[_idx].State
  OF
    E_STATION_STATE.STATION_DISABLE:
      _wStateDisable        := BitSet(_wStateDisable,(_idx - _nStationFirst));
      _wStateEnable         := BitDel(_wStateEnable, (_idx - _nStationFirst));
      _wStateOut            := BitDel(_wStateOut,    (_idx - _nStationFirst));
      _wStateGone           := BitDel(_wStateGone,   (_idx - _nStationFirst));
 
    E_STATION_STATE.STATION_ENABLE,
    E_STATION_STATE.STATION_DETECT_MOVER:
      _wStateDisable        := BitDel(_wStateDisable,(_idx - _nStationFirst));
      _wStateEnable         := BitSet(_wStateEnable, (_idx - _nStationFirst));

    E_STATION_STATE.STATION_MOVER_ENTER:
      _wStateEnable         := BitSet(_wStateEnable, (_idx - _nStationFirst));
      _wStateEnter          := BitSet(_wStateEnter,  (_idx - _nStationFirst));

    E_STATION_STATE.STATION_PROCESS_START:
      _wStateStart          := BitSet(_wStateStart,  (_idx - _nStationFirst));
      _wStateNest           := BitDel(_wStateNest,   (_idx - _nStationFirst));

    E_STATION_STATE.STATION_PROCESS_DONE:
      _wStateDone           := BitSet(_wStateDone,   (_idx - _nStationFirst));

    E_STATION_STATE.STATION_CHECK_NEST:
      _wStateStart          := BitDel(_wStateStart,  (_idx - _nStationFirst));
      _wStateDone           := BitDel(_wStateDone,   (_idx - _nStationFirst));
      _wStateNest           := BitSet(_wStateNest,   (_idx - _nStationFirst));

    E_STATION_STATE.STATION_MOVER_OUT:
      _wStateDone           := BitSet(_wStateDone,   (_idx - _nStationFirst));
      _wStateOut            := BitSet(_wStateOut,    (_idx - _nStationFirst));

    E_STATION_STATE.STATION_MOVER_GONE:
      _wStateDisable        := BitDel(_wStateDisable,(_idx - _nStationFirst));
      _wStateEnable         := BitDel(_wStateEnable, (_idx - _nStationFirst));
      _wStateEnter          := BitDel(_wStateEnter,  (_idx - _nStationFirst));
      _wStateStart          := BitDel(_wStateStart,  (_idx - _nStationFirst));
      _wStateDone           := BitDel(_wStateDone,   (_idx - _nStationFirst));
      _wStateNest           := BitDel(_wStateNest,   (_idx - _nStationFirst));
      _wStateOut            := BitDel(_wStateOut,    (_idx - _nStationFirst));

      _wStateGone           := BitSet(_wStateGone, (_idx - _nStationFirst));

    E_STATION_STATE.STATION_ERROR_LIST_STATION_ID_WRONG,  // wrong station ID in mover ticket (nTargetId written by preceeding station/process)
    E_STATION_STATE.STATION_ERROR_OUTFEED_TARGET_INVALID, // write correct target on station Ctrl.nTargetStation
    E_STATION_STATE.STATION_ERROR_INFEED_ERROR,           // clear mover error via Ctrl/State interface and retry on XTS station directly
    E_STATION_STATE.STATION_ERROR_OUTFEED_ERROR:          // clear mover error via Ctrl/State interface and retry on XTS station directly
      _wError               := BitSet(_wError,     (_idx - _nStationFirst));

    E_STATION_STATE.STATION_ERROR_FATAL:
      _wErrorFatal          := BitSet(_wErrorFatal,(_idx - _nStationFirst));

  END_CASE
END_FOR

//-----------------------------------------------------------------------------
// Mover per Minute counter all XtsStations in range
//-----------------------------------------------------------------------------
_nMoverCountTotal           :=
_AllStationMoverPerMinute   := 0; 
//-----------------------------------------------------------------------------
// mover counter
//-----------------------------------------------------------------------------
FOR _k := _nStationLast TO _nStationFirst BY(-1)
DO
  _rtrigProcess[_k](CLK:= ( _stStationCtrl[_k].Cmd = E_STATION_CTRL.STATION_MOVER_OUT));

  IF _rtrigProcess[_k].Q
  THEN
    _nMoverCount[_k]        := _nMoverCount[_k] + 1;

    IF (_MessageLevel > E_MessageType.eMessageVerbose)
    THEN
      _stMsg.eType          := E_MessageType.eMessageSentient;
      _stMsg.eDevice        := e_Device.MetricsXts + TO_UINT(_nProcessId);
                            
      _stMsg.eSubdevice     := e_Subdevice.Process_StationCollector;
      _stMsg.iErrorNumber   := _k;
      _stMsg.sText          := concat('MoverCountStation[ ]: ', TO_STRING(_nMoverCount[_k]));
      _stMsg.sText          := concat(_stMsg.sText, ': E_STATION_CTRL.');
      _stMsg.sText          := concat(_stMsg.sText, TO_STRING(_stStationCtrl[_k].Cmd));
      f_MessageSet(_stMsg);
    END_IF
  END_IF

  _rtrigProcessStart[_k](CLK:= ( _stStationState[_k].State = E_STATION_STATE.STATION_PROCESS_START));

  IF _rtrigProcessStart[_k].Q
  THEN
    _nMoverCountStart[_k]   := _nMoverCountStart[_k] + 1;

    IF (_MessageLevel > E_MessageType.eMessageVerbose)
    THEN
      _stMsg.eType          := E_MessageType.eMessageSentient;
      _stMsg.eDevice        := e_Device.MetricsXts + TO_UINT(_nProcessId);
                            
      _stMsg.eSubdevice     := e_Subdevice.Process_StationCollector;
      _stMsg.iErrorNumber   := _k;
      _stMsg.sText          := concat('MoverCountStation[ ]: ', TO_STRING(_nMoverCountEnter[_k]));
      _stMsg.sText          := concat(_stMsg.sText, ': E_STATION_STATE.');
      _stMsg.sText          := concat(_stMsg.sText, TO_STRING(_stStationState[_k].State));
      f_MessageSet(_stMsg);
    END_IF
  END_IF

  _rtrigProcessEnter[_k](CLK:= ( _stStationCtrl[_k].Cmd = E_STATION_CTRL.STATION_MOVER_ENTER));

  IF _rtrigProcessEnter[_k].Q
  THEN
    _nMoverCountEnter[_k]   := _nMoverCountEnter[_k] + 1;

    IF (_MessageLevel > E_MessageType.eMessageVerbose)
    THEN
      _stMsg.eType          := E_MessageType.eMessageSentient;
      _stMsg.eDevice        := e_Device.MetricsXts + TO_UINT(_nProcessId);
                            
      _stMsg.eSubdevice     := e_Subdevice.Process_StationCollector;
      _stMsg.iErrorNumber   := _k;
      _stMsg.sText          := concat('MoverCountStation[ ]: ', TO_STRING(_nMoverCountEnter[_k]));
      _stMsg.sText          := concat(_stMsg.sText, ': E_STATION_CTRL.');
      _stMsg.sText          := concat(_stMsg.sText, TO_STRING(_stStationCtrl[_k].Cmd));
      f_MessageSet(_stMsg);
    END_IF
  END_IF

  
  IF _tonPartsperMinute.Q
  THEN
    // count every XtsStation in range
    _nMoverPerMinute[_k]    := _nMoverCount[_k] - _nMoverCountOld[_k];
    _nMoverCountOld [_k]    := _nMoverCount[_k];

    _nMoverCountEnterOld [_k]    := _nMoverCountEnter[_k];
    _nMoverCountStartOld [_k]    := _nMoverCountStart[_k];
  END_IF
  // sum up all XtsStations in range
  _AllStationMoverPerMinute := _AllStationMoverPerMinute + _nMoverPerMinute[_k]; 
  _interAllStationsCounter  := _AllStationMoverPerMinute + _nMoverPerMinute[_k];

  // sum up all mover counts in range
  _nMoverCountTotal         := _nMoverCountTotal + _nMoverCount[_k];
END_FOR

IF _tonPartsperMinute.q
THEN
  _tonPartsperMinute(IN:=FALSE);

  IF (_MessageLevel > E_MessageType.eMessageError)
  THEN
    _stMsg.eType            := E_MessageType.eMessageBatch;
    _stMsg.eDevice          := e_Device.MetricsXts + TO_UINT(_nProcessId);
  
    _stMsg.eSubdevice       := e_Subdevice.Process_StationCollector;
    _stMsg.iErrorNumber     := _nMoverCountTotal;
    _stMsg.sText            := concat('MoverCountTotal: ', TO_STRING(_nMoverCountTotal));
    _stMsg.sText            := concat(_stMsg.sText, ': StationLast: ');
    _stMsg.sText            := concat(_stMsg.sText, TO_STRING(_nStationLast));
    _stMsg.sText            := concat(_stMsg.sText, ': StationFirst: ');
    _stMsg.sText            := concat(_stMsg.sText, TO_STRING(_nStationFirst));
    f_MessageSet(_stMsg);
  END_IF
END_IF

_tonPartsperMinute(IN:= TRUE, PT:= T#60S);
END_METHOD

PROPERTY StationCount : UINT
GET
_nStationCount    := _nStationLast - _nStationFirst + 1;
StationCount      := _nStationCount;
END_GET
END_PROPERTY

PROPERTY StationCtrl : reference to ARRAY[1..MAX_STATION] OF ST_STATION_CTRL
SET
_stStationCtrl ref= StationCtrl;
END_SET
END_PROPERTY

PROPERTY StationFirst : uint
GET
StationFirst := _nStationFirst;
END_GET
SET
_nStationFirst := StationFirst;
END_SET
END_PROPERTY

PROPERTY StationLast : uint
GET
StationLast := _nStationLast;
END_GET
SET
_nStationLast := StationLast;
END_SET
END_PROPERTY

PROPERTY StationState : reference to ARRAY[1..MAX_STATION] OF ST_STATION_STATE
SET
_stStationState REF= StationState;
END_SET
END_PROPERTY

METHOD To_T_Process : T_PROCESS // maps (2^nExp)-1 onto T_PROCESS datatype 
VAR_INPUT
  nExp              : BYTE;
END_VAR
VAR
  rVal              : LREAL;
  nTmp              : ULINT; 
  wTmp              : T_PROCESS;
END_VAR
rVal   := TO_LREAL(SEL(nExp > SIZEOF(T_PROCESS)*8, nExp, SIZEOF(T_PROCESS)*8));
nTmp   := TO_ULINT(EXPT(2,rVal)-1);

memcpy(ADR(wtmp), ADR(ntmp), SIZEOF(wtmp));

To_T_Process      := wtmp;
END_METHOD

END_FUNCTION_BLOCK

// ---- APPLICATION/_types/LinkedList/fb_Process_LinkedListCtrl.TcPOU
//---------------------------------------------------------------------------------------------------------------
//
//  HAUD 2025.12.29
//
//  - fb_LinkedListCtrl
//  -----------------------------
//  - cyclic wrapper composing fb_LinkedList
//  - used to send tickets over the mapping interfaces
//  . Ctrl / State for you to use
//---------------------------------------------------------------------------------------------------------------
FUNCTION_BLOCK fb_Process_LinkedListCtrl
VAR
  _eCheck             : E_LIST_CHECK;
  _eInit              : E_PROGRESS;

  _eCmd,
  _eCmdOld            : E_LIST_CTRL;
  _eState             : E_LIST_STATE;
  _eResult            : e_progress;

  _ItfList            : I_Process_LinkedList;

  _stCtrl             : REFERENCE TO ST_LIST_CTRL;
  _stState            : REFERENCE TO ST_LIST_STATE;

  _stNodeDataInput    : REFERENCE TO ST_LIST_NODE_DATA;   // datafield for you to write(add) your data
  _stNodeDataOutput   : REFERENCE TO ST_LIST_NODE_DATA;   // datafield for you to read (get) your data

  _stNodeDataProcess  : ST_LIST_NODE_DATA;                // local copy of ProcessData

  _stMsg              : ST_Message;
  _eDevice            : e_Device    := e_device.ProcessListCtrl;     // message device identifier
  _MessageLevel       : E_MessageType;

END_VAR

IF NOT Check() 
THEN
  _eInit                          := E_PROGRESS.PROGRESS_INVALID;
  RETURN; 
END_IF


_eCmd                           := _stCtrl.Cmd;
// check for command change
// get state for cmd
IF (_eCmd <> _eCmdOld)
THEN
  _eState                       := Cmd(_eCmd);
  _eCmdOld                      := _eCmd;

  IF (_MessageLevel > E_MessageType.eMessageError)
  THEN
    _stMsg.eType                := E_MessageType.eMessageInfo;
    _stMsg.eSubdevice           := e_Subdevice.Process_LinkedList_Com;
    _stMsg.iErrorNumber         := 0;
    _stMsg.sText                := concat(TO_STRING(_eCmd), ': ');
    _stMsg.sText                := concat(_stMsg.sText,  TO_STRING(_eState));
    f_MessageSet(_stMsg);
  END_IF
END_IF

CASE _eResult
OF
  E_PROGRESS.PROGRESS_INVALID:
    _stState.State              := TO_UINT(_eResult);

  E_PROGRESS.PROGRESS_ERROR:
    _stState.State              := _eState + E_PROGRESS.PROGRESS_ERROR;

  E_PROGRESS.PROGRESS_DONE:
    _stState.State              := _eState + E_PROGRESS.PROGRESS_DONE;

ELSE
  _stState.State                := _eState + _eResult;

  CASE _eState
  OF
    E_LIST_STATE.LIST_STATE_NULL:
      _eResult                  := E_PROGRESS.PROGRESS_DONE;

    E_LIST_STATE.LIST_STATE_INIT:
      _eResult := _eInit        := ListInit (TRUE);

    E_LIST_STATE.LIST_STATE_GET_HEAD:
      _eResult                  := ListGetHead(TRUE);

    E_LIST_STATE.LIST_STATE_GET_TAIL:
      _eResult                  := ListGetTail(TRUE);

    E_LIST_STATE.LIST_STATE_ADD_HEAD:
      _eResult                  := ListAddHead(TRUE);

    E_LIST_STATE.LIST_STATE_ADD_TAIL:
      _eResult                  := ListAddTail(TRUE);

    E_LIST_STATE.LIST_STATE_DEL_HEAD:
      _eResult                  := ListDelHead(TRUE);

    E_LIST_STATE.LIST_STATE_DEL_TAIL:
      _eResult                  := ListDelTail(TRUE);

  ELSE
    _eResult                    := E_PROGRESS.PROGRESS_INVALID;
  END_CASE
END_CASE

_stState.Count                  := _ItfList.Count;
_stState.Free                   := _ItfList.Free;
_stState.Init                   := _eInit;

METHOD Check : bool

IF NOT __ISVALIDREF(_stCtrl)
THEN
  _eCheck                     := E_LIST_CHECK.REFERENCE_CTRL_INVALID;
  RETURN;
END_IF

IF NOT __ISVALIDREF(_stState)
THEN
  _eCheck                     := E_LIST_CHECK.REFERENCE_STATE_INVALID;
  RETURN;
END_IF

IF NOT __ISVALIDREF(_stNodeDataInput)
THEN
  _eCheck                     := E_LIST_CHECK.REFERENCE_DATA_INPUT_INVALID;
  RETURN;
END_IF

IF NOT __ISVALIDREF(_stNodeDataOutput)
THEN
  _eCheck                     := E_LIST_CHECK.REFERENCE_DATA_OUTPUT_INVALID;
  RETURN;
END_IF


_eCheck                       := E_LIST_CHECK.CHECK_DONE;
Check                         := TRUE;
END_METHOD

METHOD Cmd    : E_LIST_STATE;
VAR_INPUT
  Command     : E_LIST_CTRL;
END_VAR
VAR_INST
  _eRslt      : e_progress;
  _eSt        : E_LIST_STATE;
END_VAR
IF NOT Check() THEN RETURN; END_IF

CASE Command
OF
  E_LIST_CTRL.LIST_CTRL_NULL:  // clear all method calls
    _eSt                      := E_LIST_STATE.LIST_STATE_NULL;
    _eResult                  := E_PROGRESS.PROGRESS_INIT;
    _eRslt                    := ListInit    (FALSE);
    _eRslt                    := ListAddHead (FALSE);
    _eRslt                    := ListAddTail (FALSE);
    _eRslt                    := ListDelHead (FALSE);
    _eRslt                    := ListDelTail (FALSE);
    _eRslt                    := ListGetHead (FALSE);
    _eRslt                    := ListGetTail (FALSE);

  E_LIST_CTRL.LIST_CTRL_INIT:  // clear method for initialization
    _eSt                      := E_LIST_STATE.LIST_STATE_INIT;
    _eResult := _eInit        := ListInit (FALSE);

ELSE
  IF NOT (_eInit = E_PROGRESS.PROGRESS_DONE)
  THEN
    // no init, no further commands possible
    _eSt                      := E_LIST_STATE.LIST_STATE_INVALID;

    _stMsg.eType              := E_MessageType.eMessageWarning;
    _stMsg.eSubdevice         := e_Subdevice.Process_LinkedList_Com_Cmd;
    _stMsg.iErrorNumber       := Command;
    _stMsg.sText              := concat('_eInit: ', TO_STRING(_eInit));
    _stMsg.sText              := concat(_stMsg.sText, ': ');
    _stMsg.sText              := concat(_stMsg.sText, TO_STRING(_eSt));
    f_MessageSet(_stMsg);

  ELSE
    CASE Command
    OF
      E_LIST_CTRL.LIST_CTRL_GET_HEAD:
        _eSt                  := E_LIST_STATE.LIST_STATE_GET_HEAD;
        _eResult              := ListGetHead(FALSE);

      E_LIST_CTRL.LIST_CTRL_GET_TAIL:
        _eSt                  := E_LIST_STATE.LIST_STATE_GET_TAIL;
        _eResult              := ListGetTail(FALSE);

      E_LIST_CTRL.LIST_CTRL_ADD_HEAD:
        _eSt                  := E_LIST_STATE.LIST_STATE_ADD_HEAD;
        _stNodeDataProcess      := _stNodeDataInput;
        _eResult              := ListAddHead(FALSE);

      E_LIST_CTRL.LIST_CTRL_ADD_TAIL:
        _eSt                  := E_LIST_STATE.LIST_STATE_ADD_TAIL;
        _stNodeDataProcess      := _stNodeDataInput;
        _eResult              := ListAddTail(FALSE);

      E_LIST_CTRL.LIST_CTRL_DEL_HEAD:
        _eSt                  := E_LIST_STATE.LIST_STATE_DEL_HEAD;
        _eResult              := ListDelHead(FALSE);

      E_LIST_CTRL.LIST_CTRL_DEL_TAIL:
        _eSt                  := E_LIST_STATE.LIST_STATE_DEL_TAIL;
        _eResult              := ListDelTail(FALSE);

    ELSE
        _eSt                  := E_LIST_STATE.LIST_STATE_INVALID;

        _stMsg.eType          := E_MessageType.eMessageError;
        _stMsg.eSubdevice     := e_Subdevice.Process_LinkedList_Com_Cmd;
        _stMsg.iErrorNumber   := Command;
        _stMsg.sText          := concat('Command: ', TO_STRING(Command));
        _stMsg.sText          := concat(_stMsg.sText, ': ');
        _stMsg.sText          := concat(_stMsg.sText, TO_STRING(_eSt));
        f_MessageSet(_stMsg);
    END_CASE
  END_IF
END_CASE

Cmd                           := _eSt;
END_METHOD

PROPERTY Ctrl : REFERENCE TO ST_LIST_CTRL
SET
_stCtrl ref= Ctrl;
END_SET
END_PROPERTY

PROPERTY ItfList : I_Process_LinkedList
SET
_ItfList := ItfList;
END_SET
END_PROPERTY

METHOD ListAddHead  : e_progress
VAR_INPUT
  Execute           : BOOL;
END_VAR
VAR_INST
  _ListResult       : ST_PROCESS_LIST_RESULT;
  _nErrorId         : UDINT;
  _eState           : E_PROGRESS;
END_VAR
//-----------------------------------------------------------------------------
IF NOT Execute 
THEN 
	_eState                       := E_PROGRESS.PROGRESS_INIT; 
END_IF 
//-----------------------------------------------------------------------------
IF NOT Check() 
THEN 
	ListAddHead                   := E_PROGRESS.PROGRESS_ERROR; 
	RETURN; 
END_IF
//-----------------------------------------------------------------------------
//-----------------------------------------------------------------------------
CASE _eState
OF
  E_PROGRESS.PROGRESS_INIT:
    IF Execute
    THEN
      _nErrorId                 := 0;
      _eState                   := E_PROGRESS.PROGRESS_BUSY;
    END_IF
END_CASE
//-----------------------------------------------------------------------------
//-----------------------------------------------------------------------------
CASE _eState
OF
  E_PROGRESS.PROGRESS_BUSY:
    _eState                     := E_PROGRESS.PROGRESS_PREPARE;
    _ListResult                 := _ItfList.AddHeadValue(_stNodeDataProcess.ProcessData);
END_CASE
//-----------------------------------------------------------------------------
//-----------------------------------------------------------------------------
CASE _eState
OF
  E_PROGRESS.PROGRESS_PREPARE:

    IF (_ListResult.wState <> 0)
    THEN
      _eState                   := E_PROGRESS.PROGRESS_ERROR;
      _nErrorId                 := _ListResult.wState;

      _stMsg.eType              := E_MessageType.eMessageError;
      _stMsg.eSubdevice         := e_Subdevice.Process_LinkedList_Com_AddHead;
      _stMsg.iErrorNumber       := _nErrorId;
      _stMsg.sText              := '';
      _stMsg.sText              := concat(_stMsg.sText, TO_STRING(_eState));
      f_MessageSet(_stMsg);

    ELSE
      _eState                   := E_PROGRESS.PROGRESS_DONE;

      IF (_MessageLevel > E_MessageType.eMessageError)
      THEN
        _stMsg.eType            := E_MessageType.eMessageInfo;
        _stMsg.eSubdevice       := e_Subdevice.Process_LinkedList_Com_AddHead;
        _stMsg.iErrorNumber     := 0;
        _stMsg.sText            := '';
        _stMsg.sText            := concat(_stMsg.sText, TO_STRING(_eState));
        f_MessageSet(_stMsg);
      END_IF
    END_IF
END_CASE
//-----------------------------------------------------------------------------
//-----------------------------------------------------------------------------

ListAddHead                     := _eState;
END_METHOD

METHOD ListAddTail  : e_progress
VAR_INPUT
  Execute           : BOOL;
END_VAR
VAR_INST
  _ListResult       : ST_PROCESS_LIST_RESULT;
  _nErrorId         : UDINT;
  _eState           : E_PROGRESS;
END_VAR
//-----------------------------------------------------------------------------
IF NOT Execute 
THEN 
	_eState                       := E_PROGRESS.PROGRESS_INIT; 
END_IF 
//-----------------------------------------------------------------------------
IF NOT Check() 
THEN 
	ListAddTail                   := E_PROGRESS.PROGRESS_ERROR; 
	RETURN; 
END_IF
//-----------------------------------------------------------------------------
//-----------------------------------------------------------------------------
CASE _eState
OF
  E_PROGRESS.PROGRESS_INIT:
    IF Execute
    THEN
      _nErrorId                 := 0;
      _eState                   := E_PROGRESS.PROGRESS_BUSY;
    END_IF
END_CASE
//-----------------------------------------------------------------------------
//-----------------------------------------------------------------------------
CASE _eState
OF
  E_PROGRESS.PROGRESS_BUSY:
    _eState                     := E_PROGRESS.PROGRESS_PREPARE;
    _ListResult                 := _ItfList.AddTailValue(_stNodeDataProcess.ProcessData);
END_CASE
//-----------------------------------------------------------------------------
//-----------------------------------------------------------------------------
CASE _eState
OF
  E_PROGRESS.PROGRESS_PREPARE:

    IF (_ListResult.wState <> 0)
    THEN
      _eState                   := E_PROGRESS.PROGRESS_ERROR;
      _nErrorId                 := _ListResult.wState;

      _stMsg.eType              := E_MessageType.eMessageError;
      _stMsg.eSubdevice         := e_Subdevice.Process_LinkedList_Com_AddTail;
      _stMsg.iErrorNumber       := _nErrorId;
      _stMsg.sText              := '';
      _stMsg.sText              := concat(_stMsg.sText, TO_STRING(_eState));
      f_MessageSet(_stMsg);

    ELSE
      _eState                   := E_PROGRESS.PROGRESS_DONE;

      IF (_MessageLevel > E_MessageType.eMessageError)
      THEN
        _stMsg.eType            := E_MessageType.eMessageInfo;
        _stMsg.eSubdevice       := e_Subdevice.Process_LinkedList_Com_AddTail;
        _stMsg.iErrorNumber     := 0;
        _stMsg.sText            := '';
        _stMsg.sText            := concat(_stMsg.sText, TO_STRING(_eState));
        f_MessageSet(_stMsg);
      END_IF
    END_IF
END_CASE
//-----------------------------------------------------------------------------
//-----------------------------------------------------------------------------

ListAddTail                     := _eState;
END_METHOD

METHOD ListDelHead  : e_progress
VAR_INPUT
  Execute           : BOOL;
END_VAR
VAR_INST
  _ListResult       : ST_PROCESS_LIST_RESULT;
  _nErrorId         : UDINT;
  _eState           : E_PROGRESS;
END_VAR
//-----------------------------------------------------------------------------
IF NOT Execute 
THEN 
	_eState                       := E_PROGRESS.PROGRESS_INIT; 
END_IF 
//-----------------------------------------------------------------------------
IF NOT Check() 
THEN 
	ListDelHead                   := E_PROGRESS.PROGRESS_ERROR; 
	RETURN; 
END_IF
//-----------------------------------------------------------------------------
//-----------------------------------------------------------------------------
CASE _eState
OF
  E_PROGRESS.PROGRESS_INIT:
    IF Execute
    THEN
      _nErrorId                 := 0;
      _eState                   := E_PROGRESS.PROGRESS_BUSY;
    END_IF
END_CASE
//-----------------------------------------------------------------------------
//-----------------------------------------------------------------------------
CASE _eState
OF
  E_PROGRESS.PROGRESS_BUSY:
    _eState                     := E_PROGRESS.PROGRESS_PREPARE;
    _ListResult                 := _ItfList.RemoveHeadValue();
END_CASE
//-----------------------------------------------------------------------------
//-----------------------------------------------------------------------------
CASE _eState
OF
  E_PROGRESS.PROGRESS_PREPARE:

    IF (_ListResult.wState <> 0)
    THEN
      _eState                   := E_PROGRESS.PROGRESS_ERROR;
      _nErrorId                 := _ListResult.wState;

      _stMsg.eType              := E_MessageType.eMessageError;
      _stMsg.eSubdevice         := e_Subdevice.Process_LinkedList_Com_DelHead;
      _stMsg.iErrorNumber       := _nErrorId;
      _stMsg.sText              := '';
      _stMsg.sText              := concat(_stMsg.sText, TO_STRING(_eState));
      f_MessageSet(_stMsg);

    ELSE
      _eState                   := E_PROGRESS.PROGRESS_DONE;

      IF (_MessageLevel > E_MessageType.eMessageError)
      THEN
        _stMsg.eType            := E_MessageType.eMessageInfo;
        _stMsg.eSubdevice       := e_Subdevice.Process_LinkedList_Com_DelHead;
        _stMsg.iErrorNumber     := 0;
        _stMsg.sText            := '';
        _stMsg.sText            := concat(_stMsg.sText, TO_STRING(_eState));
        f_MessageSet(_stMsg);
      END_IF
    END_IF
END_CASE
//-----------------------------------------------------------------------------
//-----------------------------------------------------------------------------

ListDelHead                     := _eState;
END_METHOD

METHOD ListDelTail  : e_progress
VAR_INPUT
  Execute           : BOOL;
END_VAR
VAR_INST
  _ListResult       : ST_PROCESS_LIST_RESULT;
  _nErrorId         : UDINT;
  _eState           : E_PROGRESS;
END_VAR
//-----------------------------------------------------------------------------
IF NOT Execute 
THEN 
	_eState                       := E_PROGRESS.PROGRESS_INIT; 
END_IF 
//-----------------------------------------------------------------------------
IF NOT Check() 
THEN 
	ListDelTail                   := E_PROGRESS.PROGRESS_ERROR; 
	RETURN; 
END_IF
//-----------------------------------------------------------------------------
//-----------------------------------------------------------------------------
CASE _eState
OF
  E_PROGRESS.PROGRESS_INIT:
    IF Execute
    THEN
      _nErrorId                 := 0;
      _eState                   := E_PROGRESS.PROGRESS_BUSY;
    END_IF
END_CASE
//-----------------------------------------------------------------------------
//-----------------------------------------------------------------------------
CASE _eState
OF
  E_PROGRESS.PROGRESS_BUSY:
    _eState                     := E_PROGRESS.PROGRESS_PREPARE;
    _ListResult                 := _ItfList.RemoveTailValue();
END_CASE
//-----------------------------------------------------------------------------
//-----------------------------------------------------------------------------
CASE _eState
OF
  E_PROGRESS.PROGRESS_PREPARE:

    IF (_ListResult.wState <> 0)
    THEN
      _eState                   := E_PROGRESS.PROGRESS_ERROR;
      _nErrorId                 := _ListResult.wState;

      _stMsg.eType              := E_MessageType.eMessageError;
      _stMsg.eSubdevice         := e_Subdevice.Process_LinkedList_Com_DelTail;
      _stMsg.iErrorNumber       := _nErrorId;
      _stMsg.sText              := '';
      _stMsg.sText              := concat(_stMsg.sText, TO_STRING(_eState));
      f_MessageSet(_stMsg);

    ELSE
      _eState                   := E_PROGRESS.PROGRESS_DONE;

      IF (_MessageLevel > E_MessageType.eMessageError)
      THEN
        _stMsg.eType            := E_MessageType.eMessageInfo;
        _stMsg.eSubdevice       := e_Subdevice.Process_LinkedList_Com_DelTail;
        _stMsg.iErrorNumber     := 0;
        _stMsg.sText            := '';
        _stMsg.sText            := concat(_stMsg.sText, TO_STRING(_eState));
        f_MessageSet(_stMsg);
      END_IF
    END_IF
END_CASE
//-----------------------------------------------------------------------------
//-----------------------------------------------------------------------------

ListDelTail                     := _eState;
END_METHOD

METHOD ListGetHead  : e_progress
VAR_INPUT
  Execute           : BOOL;
END_VAR
VAR_INST
  _ListResult       : ST_PROCESS_LIST_RESULT;
  _nErrorId         : UDINT;
  _eState           : E_PROGRESS;
END_VAR
//-----------------------------------------------------------------------------
IF NOT Execute 
THEN 
	_eState                         := E_PROGRESS.PROGRESS_INIT; 
END_IF 
//-----------------------------------------------------------------------------
IF NOT Check() 
THEN 
	ListGetHead                     := E_PROGRESS.PROGRESS_ERROR; 
	RETURN; 
END_IF
//-----------------------------------------------------------------------------
//-----------------------------------------------------------------------------
CASE _eState
OF
  E_PROGRESS.PROGRESS_INIT:
    IF Execute
    THEN
      _nErrorId                   := 0;
      _eState                     := E_PROGRESS.PROGRESS_BUSY;
    END_IF
END_CASE
//-----------------------------------------------------------------------------
//-----------------------------------------------------------------------------
CASE _eState
OF
  E_PROGRESS.PROGRESS_BUSY:
    _eState                       := E_PROGRESS.PROGRESS_PREPARE;
    _ListResult                   := _ItfList.GetHead();
END_CASE
//-----------------------------------------------------------------------------
//-----------------------------------------------------------------------------
CASE _eState
OF
  E_PROGRESS.PROGRESS_PREPARE:

    IF (_ListResult.wState <> 0)
    THEN
      _eState                     := E_PROGRESS.PROGRESS_ERROR;
      _nErrorId                   := _ListResult.wState;

      _stMsg.eType                := E_MessageType.eMessageError;
      _stMsg.eSubdevice           := e_Subdevice.Process_LinkedList_Com_GetHead;
      _stMsg.iErrorNumber         := _nErrorId;
      _stMsg.sText                := '';
      _stMsg.sText                := concat(_stMsg.sText, TO_STRING(_eState));
      f_MessageSet(_stMsg);

    ELSE
      _stNodeDataProcess.ProcessData:= _ListResult.stData;
      _stNodeDataOutput             := _stNodeDataProcess;

      _eState                     := E_PROGRESS.PROGRESS_DONE;

      IF (_MessageLevel > E_MessageType.eMessageError)
      THEN
        _stMsg.eType              := E_MessageType.eMessageInfo;
        _stMsg.eSubdevice         := e_Subdevice.Process_LinkedList_Com_GetHead;
        _stMsg.iErrorNumber       := 0;
        _stMsg.sText              := '';
        _stMsg.sText              := concat(_stMsg.sText, TO_STRING(_eState));
        f_MessageSet(_stMsg);
      END_IF
    END_IF
END_CASE
//-----------------------------------------------------------------------------
//-----------------------------------------------------------------------------

ListGetHead                       := _eState;
END_METHOD

METHOD ListGetTail  : e_progress
VAR_INPUT
  Execute           : BOOL;
END_VAR
VAR_INST
  _ListResult       : ST_PROCESS_LIST_RESULT;
  _nErrorId         : UDINT;
  _eState           : E_PROGRESS;
END_VAR
//-----------------------------------------------------------------------------
IF NOT Execute 
THEN 
	_eState                         := E_PROGRESS.PROGRESS_INIT; 
END_IF 
//-----------------------------------------------------------------------------
IF NOT Check() 
THEN 
	ListGetTail                     := E_PROGRESS.PROGRESS_ERROR; 
	RETURN; 
END_IF
//-----------------------------------------------------------------------------
//-----------------------------------------------------------------------------
CASE _eState
OF
  E_PROGRESS.PROGRESS_INIT:
    IF Execute
    THEN
      _nErrorId                   := 0;
      _eState                     := E_PROGRESS.PROGRESS_BUSY;
    END_IF
END_CASE
//-----------------------------------------------------------------------------
//-----------------------------------------------------------------------------
CASE _eState
OF
  E_PROGRESS.PROGRESS_BUSY:
    _eState                       := E_PROGRESS.PROGRESS_PREPARE;
    _ListResult                   := _ItfList.GetTail();
END_CASE
//-----------------------------------------------------------------------------
//-----------------------------------------------------------------------------
CASE _eState
OF
  E_PROGRESS.PROGRESS_PREPARE:

    IF (_ListResult.wState <> 0)
    THEN
      _eState                     := E_PROGRESS.PROGRESS_ERROR;
      _nErrorId                   := _ListResult.wState;

      _stMsg.eType                := E_MessageType.eMessageError;
      _stMsg.eSubdevice           := e_Subdevice.Process_LinkedList_Com_GetTail;
      _stMsg.iErrorNumber         := _nErrorId;
      _stMsg.sText                := '';
      _stMsg.sText                := concat(_stMsg.sText, TO_STRING(_eState));
      f_MessageSet(_stMsg);

    ELSE
      _stNodeDataProcess.ProcessData:= _ListResult.stData;
      _stNodeDataOutput             := _stNodeDataProcess;

      _eState                     := E_PROGRESS.PROGRESS_DONE;

      IF (_MessageLevel > E_MessageType.eMessageError)
      THEN
        _stMsg.eType              := E_MessageType.eMessageInfo;
        _stMsg.eSubdevice         := e_Subdevice.Process_LinkedList_Com_GetTail;
        _stMsg.iErrorNumber       := 0;
        _stMsg.sText              := '';
        _stMsg.sText              := concat(_stMsg.sText, TO_STRING(_eState));
        f_MessageSet(_stMsg);
      END_IF
    END_IF
END_CASE
//-----------------------------------------------------------------------------
//-----------------------------------------------------------------------------

ListGetTail                       := _eState;
END_METHOD

METHOD ListInit  : e_progress
VAR_INPUT
  Execute           : BOOL;
END_VAR
VAR_INST
  _ListResult       : BOOL;

  _nErrorId         : UDINT;
  _eState           : E_PROGRESS;
END_VAR
//-----------------------------------------------------------------------------
IF NOT Execute 
THEN 
	_eState                       := E_PROGRESS.PROGRESS_INIT; 
END_IF 
//-----------------------------------------------------------------------------
IF NOT Check() 
THEN 
	ListInit                      := E_PROGRESS.PROGRESS_ERROR; 
	RETURN; 
END_IF
//-----------------------------------------------------------------------------
//-----------------------------------------------------------------------------
CASE _eState
OF
  E_PROGRESS.PROGRESS_INIT:
    IF Execute
    THEN
      _nErrorId                 := 0;
      _eState                   := E_PROGRESS.PROGRESS_BUSY;
    END_IF
END_CASE
//-----------------------------------------------------------------------------
//-----------------------------------------------------------------------------
CASE _eState
OF
  E_PROGRESS.PROGRESS_BUSY:
    _eState                     := E_PROGRESS.PROGRESS_PREPARE;
    _ListResult                 := _ItfList.InitList();
END_CASE
//-----------------------------------------------------------------------------
//-----------------------------------------------------------------------------
CASE _eState
OF
  E_PROGRESS.PROGRESS_PREPARE:

    IF NOT (_ListResult)
    THEN
      _eState                   := E_PROGRESS.PROGRESS_ERROR;
      _nErrorId                 := 666;

      _stMsg.eType              := E_MessageType.eMessageError;
      _stMsg.eSubdevice         := e_Subdevice.Process_LinkedList_Com_Init;
      _stMsg.iErrorNumber       := _nErrorId;
      _stMsg.sText              := '';
      _stMsg.sText              := concat(_stMsg.sText, TO_STRING(_eState));
      f_MessageSet(_stMsg);

    ELSE
      _eState                   := E_PROGRESS.PROGRESS_DONE;

      IF (_MessageLevel > E_MessageType.eMessageError)
      THEN
        _stMsg.eType            := E_MessageType.eMessageInfo;
        _stMsg.eSubdevice       := e_Subdevice.Process_LinkedList_Com_Init;
        _stMsg.iErrorNumber     := 0;
        _stMsg.sText            := '';
        _stMsg.sText            := concat(_stMsg.sText, TO_STRING(_eState));
        f_MessageSet(_stMsg);
      END_IF
    END_IF
END_CASE
//-----------------------------------------------------------------------------
//-----------------------------------------------------------------------------

ListInit                        := _eState;
END_METHOD

PROPERTY MessageLevel : e_MessageType
GET
MessageLevel := _MessageLevel;
END_GET
SET
_MessageLevel := MessageLevel;
END_SET
END_PROPERTY

PROPERTY NodeDataInput : reference to st_list_node_data
SET
_stNodeDataInput REF= NodeDataInput;
END_SET
END_PROPERTY

PROPERTY NodeDataOutput : reference to st_list_node_data
SET
_stNodeDataOutput REF= NodeDataOutput;
END_SET
END_PROPERTY

PROPERTY State : REFERENCE TO ST_LIST_STATE
SET
_stState ref= State;
END_SET
END_PROPERTY

END_FUNCTION_BLOCK

// ---- APPLICATION/_types/fb_ProcessConductor.TcPOU
//---------------------------------------------------------------------------------------------------------------
//
//  HAUD 2025.12.30
//
//  - fb_ProcessConductor
//  -----------------------------
//  - detects new entry in the cyclic linked list wrapper
//    - forwards the received entry to target instance
//
//  - Ctrl / State for you to use (uses instance ctrl/state pair)
//  - this instance has no transport process
//    - this conductor is used for sending tickets to a transport process list
//---------------------------------------------------------------------------------------------------------------
FUNCTION_BLOCK fb_ProcessConductor EXTENDS fb_Instance
VAR
  _ItfTicketList          : I_Process_LinkedList;
  _ResultTicketList       : ST_PROCESS_LIST_RESULT;

  _WriteResult            : ST_PROCESS_LIST_RESULT;   // last job written to target
  _DeleteResult           : ST_PROCESS_LIST_RESULT;   // last job executed
END_VAR

//-----------------------------------------------------------------------------
//-----------------------------------------------------------------------------
// check pointer and interface
// connect Ctrl/State to _ItfProcessCollector
// set message device identification
//-----------------------------------------------------------------------------
IF NOT Check() THEN 
  RETURN; 
END_IF
//-----------------------------------------------------------------------------
// check command
//-----------------------------------------------------------------------------
_eCmd                                 := _stInstanceCtrl[_nProcess].Cmd;
IF (_eCmd <> _eCmdOld)
THEN
  CASE _eCmd
  OF
    E_INSTANCE_CMD.INIT:
      _eStateInstance                 := E_INSTANCE_STATE.NULL;
      _eStateProgress                 := E_PROGRESS.PROGRESS_INIT;
  END_CASE
  CmdLog();
  _eCmdOld                            := _eCmd;
END_IF
//-----------------------------------------------------------------------------
//-----------------------------------------------------------------------------
// state machine for ProcessConductor work
//-----------------------------------------------------------------------------
CASE _eStateInstance
OF
  E_INSTANCE_STATE.NULL:
    // first cycle startup
    // initialize linked list, clears all entries
    IF _ItfProcessList[_nProcess].InitList()
    THEN
      _eInit                          := E_PROGRESS.PROGRESS_INVALID;
      _eStateProgress                 := E_PROGRESS.PROGRESS_INIT;
      _eStateInstance                 := E_INSTANCE_STATE.INIT;
    END_IF

  E_INSTANCE_STATE.INIT:
    //-------------------------------------------------------------------------
    CASE _eStateProgress
    OF
    // E_INSTANCE_STATE.INIT:
    //-------------------------------------------------------------------------
      E_PROGRESS.PROGRESS_ERROR:
        ;//_eStateProgress               := E_PROGRESS.PROGRESS_INIT;

    // E_INSTANCE_STATE.INIT:
    //-------------------------------------------------------------------------
      E_PROGRESS.PROGRESS_INIT:
        IF (_ItfTicketList <> 0)
        THEN
          _eStateProgress             := E_PROGRESS.PROGRESS_BUSY;
        END_IF
    // E_INSTANCE_STATE.INIT:
    //-------------------------------------------------------------------------
      E_PROGRESS.PROGRESS_BUSY:
        IF _ItfTicketList.InitList()
        THEN
          _eInit                      := E_PROGRESS.PROGRESS_DONE;

          _eStateInstance             := E_INSTANCE_STATE.DISABLED;
          _eStateProgress             := E_PROGRESS.PROGRESS_BUSY;
        ELSE
          _eStateProgress             := E_PROGRESS.PROGRESS_ERROR;
        END_IF
      END_CASE
END_CASE
//-----------------------------------------------------------------------------
// DISABLED:
//  - clear local list result data
//  - wait for enable from the outside
//-----------------------------------------------------------------------------
CASE _eStateInstance
OF
  E_INSTANCE_STATE.DISABLED:
    //-------------------------------------------------------------------------
    CASE _eStateProgress
    OF
      E_PROGRESS.PROGRESS_BUSY:
        CASE _eCmd
        OF
          E_INSTANCE_CMD.ENABLE:      // turn it on!!
            _eStateInstance           := E_INSTANCE_STATE.DETECTION;
            _eStateProgress           := E_PROGRESS.PROGRESS_BUSY;
  
            IF (_MessageLevel > E_MessageType.eMessageInfo)
            THEN
              _stMsg.eType            := E_MessageType.eMessageVerbose;
              _stMsg.eSubdevice       := e_Subdevice.Instance_ProcessConductor;
              _stMsg.iErrorNumber     := 0;
              _stMsg.sText            := concat(TO_STRING(_eStateInstance), ': ');
              _stMsg.sText            := concat(_stMsg.sText, TO_STRING(_eStateProgress));
              f_MessageSet(_stMsg);
            END_IF

        END_CASE
    END_CASE
END_CASE
//-----------------------------------------------------------------------------
// DETECTION: 
//  - check inked list and GetHead()
//  - copy job data
//  - switch on process
//-----------------------------------------------------------------------------
CASE _eStateInstance
OF
  E_INSTANCE_STATE.DETECTION:
    //-------------------------------------------------------------------------
    CASE _eStateProgress
    OF
      E_PROGRESS.PROGRESS_BUSY:
        IF (_eCmd = E_INSTANCE_CMD.DISABLE)
        THEN
          _eStateInstance             := E_INSTANCE_STATE.DISABLED;
          _eStateProgress             := E_PROGRESS.PROGRESS_INIT;

        ELSIF (_ItfTicketList.Count > 0)
        THEN
          // get new job order for my process
          _stListResult               := _ItfTicketList.GetHead();  // the list results carries information about the requirements of the target process (who and where)

          IF (_stListResult.wState <> 0)
          THEN
            // error in list results must not appear
            // if you land here, there is somethng wrong with the initialization or configuration of the linked list
            _eStateProgress           := E_PROGRESS.PROGRESS_ERROR;

            _stMsg.eType              := E_MessageType.eMessageError;
            _stMsg.eSubdevice         := e_Subdevice.Ticket_LinkedList_Com_GetHead;
            _stMsg.iErrorNumber       := _stListResult.wState;
            _stMsg.sText              := concat(TO_STRING(_eStateInstance), ': _ListResult.wState: ');
            _stMsg.sText              := concat(_stMsg.sText, TO_STRING(_eStateProgress));
            f_MessageSet(_stMsg);

          ELSE
            IF (_MessageLevel > E_MessageType.eMessageError)
            THEN
              _stMsg.eType            := E_MessageType.eMessageInfo;
              _stMsg.eSubdevice       := e_Subdevice.Ticket_LinkedList_Com_GetHead;
              _stMsg.iErrorNumber     := 0;
              _stMsg.sText            := concat(TO_STRING(_eStateInstance), ': ');
              _stMsg.sText            := concat(_stMsg.sText, '_ListResult.stData.wTarget: ');
              _stMsg.sText            := concat(_stMsg.sText, _ItfProcessCollector[_nProcess].BitsToString(_stListResult.stData.wTarget));
              f_MessageSet(_stMsg);
            END_IF

            _stProcessData            := _stListResult.stData;  // list result contains data for target process


            IF (_stProcessData.wTarget > 0)
            THEN
              _eStateProgress         := E_PROGRESS.PROGRESS_PREPARE;      // reset substate


              IF (_MessageLevel > E_MessageType.eMessageEmpty)
              THEN
                _stMsg.eType          := E_MessageType.eMessageBatch;
                _stMsg.eSubdevice     := e_Subdevice.Instance_ProcessConductor;
                _stMsg.iErrorNumber   := 0;
                _stMsg.sText          := concat(TO_STRING(_eStateProgress), ': ');
                _stMsg.sText          := concat(_stMsg.sText, TO_STRING(e_message_batch.MSG_BATCH_JOB_STARTED));
                f_MessageSet(_stMsg);
              END_IF
            ELSE
              _ResultTicketList       := _ItfTicketList.RemoveHeadValue();
            END_IF

            // check target mask for entries
            IF NOT (_stProcessData.wTarget > 0)
            THEN
              //_eStateProgress         := E_PROGRESS.PROGRESS_ERROR;

              _stMsg.eType            := E_MessageType.eMessageWarning;
              _stMsg.eSubdevice       := e_Subdevice.Process_LinkedList_CheckData;
              _stMsg.iErrorNumber     := 666;
              _stMsg.sText            := concat(TO_STRING(_eStateInstance), ': ');
              _stMsg.sText            := concat(_stMsg.sText, '_ProcessData.wTarget: ');
              _stMsg.sText            := concat(_stMsg.sText, _ItfProcessCollector[_nProcess].BitsToString(_stProcessData.wTarget));
              f_MessageSet(_stMsg);
            END_IF
          END_IF
        END_IF
    END_CASE
    CASE _eStateProgress
    OF
      E_PROGRESS.PROGRESS_PREPARE:
      // check process target plausibility
      IF NOT (_stProcessData.nProcessId > 0) OR
         NOT (_stProcessData.nProcessId < E_INSTANCE.INSTANCE_MAX)
      THEN
        _eStateProgress               := E_PROGRESS.PROGRESS_ERROR;
      ELSE
        _DeleteResult                 := _ItfTicketList.RemoveHeadValue();

        IF (_DeleteResult.wState = 0)
        THEN
          _eStateInstance             := E_INSTANCE_STATE.WORKING;      // go check if my process is switched on
          _eStateProgress             := E_PROGRESS.PROGRESS_BUSY;      // reset substate
        ELSE
          _eStateProgress             := E_PROGRESS.PROGRESS_ERROR;
        END_IF
      END_IF
    END_CASE
END_CASE
//-----------------------------------------------------------------------------
// WORKING
//  - Add ticket in target list
//  - check and log
//  - transition to finish
//-----------------------------------------------------------------------------
CASE _eStateInstance
OF
  E_INSTANCE_STATE.WORKING:
    //-------------------------------------------------------------------------
    CASE _eStateProgress
    OF
      E_PROGRESS.PROGRESS_BUSY:
        // write process ticket, then go back up
        _WriteResult                  := _ItfProcessList[_stProcessData.nProcessId].AddTailValue(_stProcessData);

        IF (_WriteResult.wState <> 0)
        THEN
          // adding to target list must be successful on the first try
          // IF you land here, there is something wrong with initialization or configuration of the linked list
          _eStateProgress             := E_PROGRESS.PROGRESS_ERROR;
        ELSE
          _eStateInstance             := E_INSTANCE_STATE.FINISH;
          _eStateProgress             := E_PROGRESS.PROGRESS_BUSY;

          IF (_MessageLevel > E_MessageType.eMessageInfo)
          THEN
            _stMsg.eType              := E_MessageType.eMessageVerbose;
            _stMsg.eSubdevice         := e_Subdevice.Process_LinkedList_AddTail;
            _stMsg.iErrorNumber       := _stProcessData.nProcessId;
            _stMsg.sText              := concat(TO_STRING(_eStateInstance), ': ');
            _stMsg.sText              := concat(_stMsg.sText, TO_STRING(_eStateProgress));
            f_MessageSet(_stMsg);
          END_IF
        END_IF
    END_CASE
END_CASE
//-----------------------------------------------------------------------------
// FINISH:
//-----------------------------------------------------------------------------
CASE _eStateInstance
OF
  E_INSTANCE_STATE.FINISH:
    //-------------------------------------------------------------------------
    CASE _eStateProgress
    OF
      E_PROGRESS.PROGRESS_BUSY:
        _eStateProgress               := E_PROGRESS.PROGRESS_DONE;
    END_CASE
    // E_INSTANCE_STATE.FINISH:
    //-------------------------------------------------------------------------
    CASE _eStateProgress
    OF
      E_PROGRESS.PROGRESS_DONE:
        CASE _eCmd
        OF
          E_INSTANCE_CMD.FINISH:
            _eStateInstance           := E_INSTANCE_STATE.DISABLED;
            _eStateProgress           := E_PROGRESS.PROGRESS_BUSY;
        END_CASE
    END_CASE
END_CASE
//-----------------------------------------------------------------------------
//-----------------------------------------------------------------------------
_stInstanceState[_nProcess].State     := _eStateInstance;
_stInstanceState[_nProcess].Progress  := _eStateProgress;
//-----------------------------------------------------------------------------
//-----------------------------------------------------------------------------
_stInstanceState[_nProcess].StationCount      := _ItfProcessCollector[_nProcess].StationCount;
_stInstanceState[_nProcess].QueueProcessCount := _ItfProcessCollector[_nProcess].QueueProcessCount;
//-----------------------------------------------------------------------------
//-----------------------------------------------------------------------------

PROPERTY TicketLinkedList : I_Process_LinkedList
SET
_ItfTicketList := TicketLinkedList;
END_SET
END_PROPERTY

END_FUNCTION_BLOCK

// ---- _XML/Configuration/fb_Configuration.TcPOU
//---------------------------------------------------------------------------------------------------------------
//
//  fb_Configuration
//
//  HAUD 2023.04.14
//  - base xml integration
//
//  HAUD 2026.04.10.
//  - now extending a base class
//
//  - cyclic OnChange wrapper for xml data 
//      - Ctrl/State
//        1. INIT
//        2. READ / WRITE
//
//  - read  ST_STATION_PARAMETER on demand
//  - write ST_STATION_PARAMETER on demand
//
//---------------------------------------------------------------------------------------------------------------
// This SOFTWARE is provided as an Example by THE PROVIDER "as is" and "with all faults." THE PROVIDER makes no 
// representations or warranties of any kind concerning the safety, suitability, lack of viruses, inaccuracies, 
// typographical errors, or other harmful components of this SOFTWARE. There are inherent dangers in the use of 
// any software, and you are solely responsible for determining whether this SOFTWARE is compatible with your 
// equipment and other software installed on your equipment. You are also solely responsible for the protection 
// of your equipment and backup of your data, and THE PROVIDER will not be liable for any damages you may suffer 
// in connection with using, modifying, or distributing this SOFTWARE.
//---------------------------------------------------------------------------------------------------------------
FUNCTION_BLOCK fb_Configuration EXTENDS fb_XmlBase
VAR
  _stCtrl               : REFERENCE TO ST_DATA_CTRL;
  _stState              : REFERENCE TO ST_DATA_STATE;

  _stConfiguration      : ST_Configuration;
  _pStationParameter    : POINTER TO ARRAY[1..MAX_STATION] OF ST_STATION_PARAMETER;
END_VAR
VAR CONSTANT
  FILE_ROOT             : STRING := 'CONFIG_XtsTransport_';
  X_PATH                : STRING := '/XtsTransport/config';
END_VAR

//---------------------------------------------------------------------------------------------------------------
//  check pointers from the outside
//---------------------------------------------------------------------------------------------------------------
IF NOT Check() THEN RETURN; END_IF
//---------------------------------------------------------------------------------------------------------------
// always build the internal data pointer
//  - as always: better safe than sorry
//  - leave this bit here, it doesn't cost much and safely addresses the data
//---------------------------------------------------------------------------------------------------------------
_pData                        := ADR    (_stConfiguration);
_nData                        := SIZEOF (_stConfiguration);
_sXpath                       := X_PATH;

// copy to local for debug
_eCmd                         := _stCtrl.Cmd;

// cyclic check for command change
// get state for cmd
IF (_eCmd <> _eCmdOld)
THEN
  // get matching sdtate for Ctrl.Cmd
  _eState                     := Cmd(_eCmd);
  _eCmdOld                    := _eCmd;
END_IF


CASE _eResult
OF
  E_PROGRESS.PROGRESS_INVALID:
    _stState.State            := E_DATA_STATE.NULL;

  E_PROGRESS.PROGRESS_ERROR:
    _stState.State            := _eState + E_PROGRESS.PROGRESS_ERROR;

  E_PROGRESS.PROGRESS_DONE:
    _stState.State            := _eState + E_PROGRESS.PROGRESS_DONE;

ELSE
  // work in progress
  // update progress for extern use
  _stState.State              := _eState + _eResult;

  CASE _eState
  OF
    E_DATA_STATE.INIT:
      _eResult   := _eInit    := CreateFolder(TRUE);

    E_DATA_STATE.READ:
      _eResult                := XmlRead(TRUE);
      IF (_eResult = E_PROGRESS.PROGRESS_DONE)
      THEN
        // copy the single ladies
        memcpy(_pStationParameter, ADR(_stConfiguration.XtsStationParameter), SIZEOF(_stConfiguration.XtsStationParameter));
      END_IF

    E_DATA_STATE.WRITE:
      _eResult                := XmlWrite(TRUE);
  ELSE
      _eResult                := E_PROGRESS.PROGRESS_INVALID;
  END_CASE
END_CASE

METHOD Check : BOOL
//-------------------------------------------------------------------------
IF NOT (__ISVALIDREF(_stCtrl))
THEN
  _eCheck               := E_DATA_CHECK.REFERENCE_CTRL_INVALID;
  RETURN;
END_IF
//-------------------------------------------------------------------------
IF NOT (__ISVALIDREF(_stState))
THEN
  _eCheck               := E_DATA_CHECK.REFERENCE_STATE_INVALID;
  RETURN;
END_IF
//-------------------------------------------------------------------------
IF NOT (_pStationParameter <> 0)
THEN
  _eCheck               := E_DATA_CHECK.POINTER_STATION_PARAMETER_INVALID;
  RETURN;
END_IF
//-------------------------------------------------------------------------
_eCheck                 := E_DATA_CHECK.DONE_CHECK;
Check                   := TRUE;
END_METHOD

METHOD PRIVATE Cmd : E_DATA_STATE
VAR_INPUT
  Ctrl      : E_DATA_CTRL;
END_VAR
VAR_INST
  _eState   : E_DATA_STATE;
END_VAR
IF NOT Check() THEN Cmd   := E_DATA_STATE.NULL;  RETURN; END_IF

CASE Ctrl
OF
  //---------------------------------------------------------------
  E_DATA_CTRL.INIT:
    _sName                := concat(FILE_ROOT, _sIdentity);
    _sName                := concat(_sName, '.xml');
    _sFilePath            := concat(_sDirectoryPath, _sName);

    _eInit                := E_PROGRESS.PROGRESS_INVALID;
    _eResult              := CreateFolder(FALSE);
    _eState               := E_DATA_STATE.INIT;
  //---------------------------------------------------------------
  E_DATA_CTRL.READ:
    _eResult              := XmlRead(FALSE);
    _eState               := E_DATA_STATE.READ;
  //---------------------------------------------------------------
  E_DATA_CTRL.WRITE:
    _stConfiguration.XtsStationParameter  := _pStationParameter^;

    _eResult              := XmlWrite(FALSE);
    _eState               := E_DATA_STATE.WRITE;
ELSE
  //---------------------------------------------------------------
    _eResult              := E_PROGRESS.PROGRESS_INVALID; 
    _eState               := E_DATA_STATE.NO_EXIST;
END_CASE

Cmd                       := _eState;
END_METHOD

PROPERTY Ctrl : REFERENCE to ST_DATA_CTRL
SET
_stCtrl ref= Ctrl;
END_SET
END_PROPERTY

